// SIMATIC STEP 7 (V5.x) project COB#1&2_GC#2_07_12_2012
// CPU: CPU 315-2 DP
// CPU: CPU 315-2 DP
// station: Hardware
// station: SIMATIC 300 - BEC
// station: P_ADR_BUS
// station: Hardware
// station: SIMATIC 300 - TATA
// station: P_ADR_BUS

SYMBOL_TABLE
"MAIN_POWER_DB"	DB 1	DB 1	// MAIN POWER DATA BLOCK
"HYDRAULIC_FUNCTIONS_DB"	DB 2	DB 2	// HYDRAULIC FUNCTIONS DB
"TRAVEL_DRIVE_DB"	DB 3	DB 3	// TRAVEL DRIVE DATA BLOCK
"AIR_COMPRESSOR_DB"	DB 4	DB 4	// AIR COMPRESSOR DATA BLOCK
"HOOD_SYSTEM_DB"	DB 5	DB 5	// HOOD SYSTEM OPERATIONS DATA BLOCK
"DOOR_EXTRACTOR_DB"	DB 6	DB 6	// DOOR EXTRACTOR MECHANISH DATA BLOCK
"SERVICE_PLATFORM_DB"	DB 7	DB 7	// SERVICE PLATFORM DATA BLOCK
"JAMB_CLEANER_DB"	DB 8	DB 8	// JAMB CLEANER DATA BLOCK
"GUIDE_CAGE_DB"	DB 9	DB 9	// GUIDE CAGE DATA BLOCK
"DOOR_CLEANER_MOTOR_DB"	DB 10	DB 10	// DOOR CLEANER MOTOR DATA BLOCK
"WIN_CC_DB"	DB 11	DB 11	// WIN CC HMI DATA BLOCK
"CMD_FROM_TATA"	DB 12	DB 12	// COMMANDS FROM TATA PLC THROUGH PROFIBUS
"FB_TO_TATA"	DB 13	DB 13	// FEEDBACK TO TATA THROUGH PROFIBUS
"TATA_COMMUNICATION_DB"	DB 14	DB 14	// TATA COMMUNICATION DATA BLOCK
"INPUT_MAPPING"	FC 1	FC 1	// INPUT MAPPING FUNCTION
"OUTPUT_MAPPING"	FC 2	FC 2	// OUTPUT MAPPING FUNCTION
"MAIN_POWER"	FC 3	FC 3	// MAIN POWER CONTROL LOGIC
"HYDRAULIC_SYSTEM"	FC 4	FC 4	// HYDRAULIC SYSTEM OPERATIONS
"TRAVEL_DRIVE"	FC 5	FC 5	// TRAVEL_DRIVE_MECHANISM
"AIR_COMPRESSOR"	FC 6	FC 6	// AIR COMPRESSOR FUNCTION
"HOOD_SYSTEM"	FC 7	FC 7	// HOOD SYSTEM OPERATIONS
"DOOR_EXTRACTOR"	FC 8	FC 8	// DOOR EXTRACTOR MECHANISM
"SERVICE_PLATFORM"	FC 9	FC 9	// SERVICE PLATFORM OPERATIONS
"JAMB_CLEANER"	FC 10	FC 10	// JAMB CLEANER FUNCTIONS
"GUIDE_CAGE"	FC 11	FC 11	// GUIDE CAGE FUNCTION
"DOOR_CLEANER_MOTOR"	FC 12	FC 12	// DOOR CLEANER MOTOR FUNCTIONS
"PROFIBUS_COMMUNICATION"	FC 13	FC 13	// PROFIBUS COMMUNICATION LOGIC
"TATA_COMMUNICATION"	FC 14	FC 14	// TATA COMMUNICATION FUNCATIONS
"SCALE"	FC 105	FC 105	// Scaling Values
"UNSCALE"	FC 106	FC 106	// Unscaling Values
"MAIN_PWR_RDY_FOR_ON"	I 0.0	BOOL	// MAIN POWER READY FOR ON
"MAIN_PWR_ON_FB"	I 0.1	BOOL	// MAIN POWER ON FEED BACK
"CTRL_PWR_ON_FB"	I 0.2	BOOL	// CONTROL POWER ON FEEDBACK
"MAIN_PWR_ON_PB"	I 0.3	BOOL	// MAIN POWER ON PUSH BUTTON
"MAIN_PWR_OFF_PB"	I 0.4	BOOL	// MAIN POWER OFF PUSH BUTTON
"LAMP_TEST_PB"	I 0.5	BOOL	// LAMP TEST PUSH BUTTON
"ALARM_ACK_PB"	I 0.6	BOOL	// ALARM ACKNOWLEDGE PUSH BUTTON
"SERVICE_PF_STP_PB"	I 0.7	BOOL	// SERVICE PLATFORM STOP PUSH BUTTON
"CTRL_SELECTION_CD"	I 1.0	BOOL	// CONTROL SELECTRION CD
"EXT_OVN_DOR_STA_PB"	I 1.1	BOOL	// EXTRACT OVEN DOOR STAT PUSH PUSH BUTTON
"RPL_OVN_DOR_STA_PB"	I 1.2	BOOL	// REPLACE OVEN DOOR STAT PUSH PUSH BUTTON
"EXT_RPL_FUNC_STP_PB"	I 1.3	BOOL	// EXTRACT AND REPLACE FUNCTION STOP PUSH BUTTON
"GC_TRA_AUTO_STA_PB"	I 1.4	BOOL	// GUIDE CAGE TRAVEL AUTO START PUSH BUTTON
"GC_TRA_AUTO_STP_PB"	I 1.5	BOOL	// GUIDE CAGE TRAVEL AUTO STOP PUSH BUTTON
"CLN_OVN_JMB_STA_PB"	I 1.6	BOOL	// CLEAN OVEN JAMB AUTO START PUSH BUTTON
"ALL_OPER_IN_REP_MODE"	I 1.7	BOOL	// ALL OPERATIONS IN REPAIR MODE
"CLN_OVN_JMB_STP_PB"	I 2.0	BOOL	// CLEAN OVEN JAMB AUTO STOP PUSH BUTTON
"ALL_MECH_QUICK_STOP"	I 2.1	BOOL	// ALL MECHANICAL OPERATIONS QUICK STOP
"CLN_OVN_DR_STA_PB"	I 2.2	BOOL	// CLEAN OVEN DOOR START PUSH BUTTON
"CLN_OVN_DR_STP_PB"	I 2.3	BOOL	// CLEAN OVEN DOOR STOP PUSH BUTTON
"CD_EMERGENCY_STOP"	I 2.4	BOOL	// CONTROL DESK EMERGENCY STOP
"SERVICE_PF_STA_PB"	I 2.5	BOOL	// SERVICE PLATFORM START PUSH BUTTON
"REP_MAN_SS"	I 2.6	BOOL	// REPAIR/MANUAL SELECTOR SWITCH
"ALL_OPER_IN_OPER_MODE"	I 2.7	BOOL	// ALL OPERATIONS IN OPERATION MODE
"JC_VC_HM_STA_PB"	I 3.0	BOOL	// JAMB CLEANER HOME START PB
"ID_FAN_READY"	I 3.1	BOOL	// ID FAN DRIVE READY FOR START
"PUMP_1_RUN_FB"	I 3.2	BOOL	// PUMP 1 RUNNING FEEDBACK
"PUMP_1_OVR_LD_TRIP"	I 3.3	BOOL	// PUMP 1 OVER LOAD TRIPPED
"PUMP_2_RDY_FOR_STA"	I 3.4	BOOL	// PUMP 2 READY FOR START
"PUMP_2_RUN_FB"	I 3.5	BOOL	// PUMP 2 RUNNING FEEDBACK
"PUMP_2_OVR_LD_TRIP"	I 3.6	BOOL	// PUMP 2 OVER LOAD TRIPPED
"CIR_PUMP_RDY_FOR_STA"	I 4.0	BOOL	// CIRCULATION PUMP READY FOR START
"CIR_PUMP_RUN_FB"	I 4.1	BOOL	// CIRCULATION PUMP RUNNING FEEDBACK
"CIR_PUMP_OVR_LD_TRIP"	I 4.2	BOOL	// CIRCULATION PUMP OVER LOAD TRIPPED
"COLR_FAN_RDY_FOR_STA"	I 4.3	BOOL	// COOLER FAN READY FOR START
"COLR_FAN_RUN_FB"	I 4.4	BOOL	// COOLER FAN RUNNING FEEDBACK
"COLR_FAN_OVR_LD_TRIP"	I 4.5	BOOL	// COOLER FAN OVER LOAD TRIPPED
"CD_LCS_SS"	I 4.6	BOOL	// CONTROL DESK / LOCAL CONTROL SELECTOR SWITCH
"PUMP_1_2_SS"	I 5.0	BOOL	// PUMP 1 OR 2 SELECTOR SWITCH
"PUMP_1_STA_PB"	I 5.1	BOOL	// PUMP 1 START PUSH BUTTON
"PUMP_1_STP_PB"	I 5.2	BOOL	// PUMP 1 STOP PUSH BUTTON
"PUMP_2_STA_PB"	I 5.3	BOOL	// PUMP 2 START PUSH BUTTON
"PUMP_2_STP_PB"	I 5.4	BOOL	// PUMP 2 STOP PUSH BUTTON
"EMERGENCY_STOP_PB"	I 5.5	BOOL	// EMERGENCY STOP PUSH BUTTON
"LAMP_TEST_PB_LCS_41"	I 5.6	BOOL	// LAMP TEST PUSH BITTON LCS 41
"SP_TRA_FWD_STA_PB"	I 5.7	BOOL	// SERVICE PLATFORM TRAVEL FORWARD PUSH BUTTON
"PUMP_1_2_SS_LCS"	I 6.0	BOOL	// PUMP 1 OR 2 SELECTOR SWITCH LCS
"PUMP_1_STA_PB_LCS"	I 6.1	BOOL	// PUMP 1 START PUSH BUTTON LCS
"PUMP_1_STP_PB_LCS"	I 6.2	BOOL	// PUMP 1 STOP PUSH BUTTON LCS
"PUMP_2_STA_PB_LCS"	I 6.3	BOOL	// PUMP 2 START PUSH BUTTON LCS
"PUMP_2_STP_PB_LCS"	I 6.4	BOOL	// PUMP 2 STOP PUSH BUTTON LCS
"CIR_PUMP_STA_PB_LCS"	I 6.5	BOOL	// CIRCULATION PUMP START PUSH BUTTON LCS
"CIR_PUMP_STP_PB_LCS"	I 6.6	BOOL	// CIRCULATION PUMP STOP PUSH BUTTON LCS
"SP_TRA_REV_STA_PB"	I 6.7	BOOL	// SERVICE PLATFORM TRAVEL REVERSE START PUSH BUTTON
"COLR_FAN_STA_PB_LCS"	I 7.0	BOOL	// COOLER FAN START PUSH BUTTON LCS
"COLR_FAN_STP_PB_LCS"	I 7.1	BOOL	// COOLER FAN STOP PUSH BUTTON LCS
"EMG_ACCM_STA_PB_LCS"	I 7.2	BOOL	// EMERGENCY ACCUMULATOR START PB LCS
"EMG_ACCM_STP_PB_LCS"	I 7.3	BOOL	// EMERGENCY ACCUMULATOR STOP PB LCS
"SHT_OF_VLV_LIN_1_FUL_OPN"	I 7.4	BOOL	// SHUT OFF VALVE IN LINE 1 - FULLY OPEN
"SHT_OF_VLV_LIN_2_FUL_OPN"	I 7.5	BOOL	// SHUT OFF VALVE IN LINE 2 - FULLY OPEN
"LOW_OIL_TEMP"	I 7.6	BOOL	// LOW OIL TEMPERATURE - THERMOSTAT
"SP_STP_PB"	I 7.7	BOOL	// SERVICE PLATFORM STOP PUSH BUTTON
"HIGH_OIL_TEMP"	I 8.0	BOOL	// HIGH OIL TEMPERATURE - THERMOSTAT
"MAX_OIL_TEMP"	I 8.1	BOOL	// MAXIMUM OIL TEMPERATURE - THERMOSTAT
"LOW_OIL_LEVEL"	I 8.2	BOOL	// LOW OIL LEVEL - FLOAT SWITCH
"MIN_OIL_LEVEL"	I 8.3	BOOL	// MINIMUM OIL LEVEL - FLOAT SWITCH
"RET_LIN_FLTR_CKD"	I 8.4	BOOL	// RETURN LINE FILTER CHOKED
"LOW_OIL_PRESS"	I 8.5	BOOL	// LOW OIL PRESSURE - PRESSURE SWITCH
"HIGH_OIL_PRESS"	I 8.6	BOOL	// HIGH OIL PRESSURE - PRESSURE SWITCH
"SP_AUTO_SS"	I 8.7	BOOL	// SERVICE PLATFORM AUTO SELECTOR SWITCH
"TRA_GRP_1_BRK_RDY_FOR_ST"	I 9.0	BOOL	// TRAVEL GROUP 1 BREAK READY FOR START
"TRA_GRP_1_BRK_ON_FB"	I 9.1	BOOL	// TRAVEL GROUP 1 BREAK ON FEEDBACK
"TRA_GRP_2_BRK_RDY_FOR_ST"	I 9.2	BOOL	// TRAVEL GROUP 2 BREAK READY FOR START
"TRA_GRP_2_BRK_ON_FB"	I 9.3	BOOL	// TRAVEL GROUP 2 BREAK ON FEEDBACK
"TRA_JOY_STK_DED_MAN_BTN"	I 9.4	BOOL	// TRAVEL JOY DEAD MAN BUTTON
"TRA_JOY_STK_HME_POS"	I 9.5	BOOL	// TRAVEL JOY STICK HOME POSITION
"TRA_JOY_STK_FWD_POS"	I 9.6	BOOL	// TRAVEL JOY STICK FOWRWARD POSITION
"TRA_JOY_STK_REV_POS"	I 9.7	BOOL	// TRAVEL JOY DEAD REVERSE POSITION
"TRA_MODE_AUTO_MAN_SS"	I 10.0	BOOL	// TRAVEL MODE AUTO/MANUAL BUTTON
"LASER_SPOTTING"	I 10.1	BOOL	// TRAVEL LASER SPOTTING
"AUTO_POS_ACK"	I 10.2	BOOL	// AUTO POSITION ACKNOWLEDGE
"TRA_DRV_1_PROF_HARD_SS"	I 10.3	BOOL	// TRAVEL DRIVE 1 PROFIBUS/HARD WIRE SELECTRO SWITCH
"TRA_DRV_1_ON_FB"	I 10.4	BOOL	// TRAVEL DRIVE 1 ON FEEDBACK
"TRA_DRV_1_RDY_FOR_STA"	I 10.5	BOOL	// TRAVEL DRIVE 1 READY FOR START
"TRA_DRV_1_TRP_FB"	I 10.6	BOOL	// TRAVEL DRIVE 1 TRIP FEEDBACK
"TRA_DRV_2_PROF_HARD_SS"	I 10.7	BOOL	// TRAVEL DRIVE 2 PROFIBUS/HARD WIRE SELECTRO SWITCH
"TRA_DRV_2_ON_FB"	I 11.0	BOOL	// TRAVEL DRIVE 2 ON FEEDBACK
"TRA_DRV_2_RDY_FOR_STA"	I 11.1	BOOL	// TRAVEL DRIVE 2 READY FOR START
"TRA_DRV_2_TRP_FB"	I 11.2	BOOL	// TRAVEL DRIVE 2 TRIP FEEDBACK
"LIMIT_SW_END_FWD_FB"	I 11.3	BOOL	// LIMIT SWITCH END FORWARD FEEDBACK
"LIMIT_SW_END_EMG_FWD_FB"	I 11.4	BOOL	// LIMIT SWITCH END FORWARD EMERGENCY FEEDBACK
"LIMIT_SW_END_REV_FB"	I 11.5	BOOL	// LIMIT SWITCH END REVERSE FEEDBACK
"LIMIT_SW_END_EMG_REV_FB"	I 11.6	BOOL	// LIMIT SWITCH END REVERSE EMERGENCY FEEDBACK
"SP_MAN_SS"	I 11.7	BOOL	// SERVICE PLATFORM MANUAL SELECTOR SWITCH
"SP_TRA_FWD_LS"	I 12.0	BOOL	// SERVICE PLATFORM TRAVEL FORWARD LIMIT SWITCH
"AC_RDY_FOR_STA"	I 12.1	BOOL	// AIR COMPRESSOR READY FOR START
"AC_RUN_FB"	I 12.2	BOOL	// AIR COMPRESSOR RUN FEED BACK
"AC_OLR_TRIP_FB"	I 12.3	BOOL	// AIR COMPRESSOR TRIP FEED BACK
"AC_STA_PB"	I 12.4	BOOL	// AIR COMPRESSOR START PUSH BUTTON
"AC_STP_PB"	I 12.5	BOOL	// AIR COMPRESSOR STOP PUSH BUTTON
"ID_FAN_PROFI_HW_SS"	I 12.6	BOOL	// ID FAN PROFIBUS/HARDWIRE CONNECTION
"SP_TRA_REV_LS"	I 12.7	BOOL	// SERVICE PLATFORM TRAVEL REVERSE LIMIT SWITCH
"ID_FAN_DRV_ON_FB"	I 13.0	BOOL	// ID FAN DRIVE ON FEEDBACK
"ID_FAN_DRV_RDY_FOR_STA"	I 13.1	BOOL	// ID FAN DRIVE READY FOR START
"ID_FAN_DRV_TRIP_FB"	I 13.2	BOOL	// ID FAN DRIVE TRIP FEED BACK
"WTR_PMP_DRV_RDY_FOR_STA"	I 13.3	BOOL	// WATER PUMP DRIVE READY FOR START
"WTR_PMP_DRV_ON_FB"	I 13.4	BOOL	// WATER PUMP DRIVE ON FEEDBACK
"WTR_PMP_DRV_TRIP_FB"	I 13.5	BOOL	// WATER PUMP DRIVE TRIP FEED BACK
"HOOD_STA_PB"	I 13.6	BOOL	// HOOD START PUSH BUTTON
"EMERGENCY_STOP_PB_PANEL"	I 13.7	BOOL	// EMERGENCY STOP PUSH BUTTON IN PLC PANEL
"HOOD_STP_PB"	I 14.0	BOOL	// HOOD STOP PUSH BUTTON
"ID_FAN_LS_HS_SEL"	I 14.1	BOOL	// ID FAN LOW SPEED/HIGH SPEED SELECTION
"WTR_LEV_LOW_LEV_SWH"	I 14.2	BOOL	// WATER LEVEL LOW LEVEL SWITCH
"SLEW_SLOW_FWD_LS"	I 14.3	BOOL	// SLEW SLOW FORWARD LIMIT SWITCH
"SLEW_SLOW_RET_LS"	I 14.4	BOOL	// SLEW SLOW RETRACT LIMIT SWITCH
"SLEW_NOR_FWD_LS"	I 14.5	BOOL	// SLEW NORMAL FORWARD LIMIT SWITCH
"SLEW_NOR_RET_LS"	I 14.6	BOOL	// SLEW NORMAL RETRACT LIMIT SWITCH
"TRA_ILK_BYPASS"	I 14.7	BOOL	// TRAVEL INTERLOCK BYPASS INPUT
"TRA_SLOW_FWD_LS"	I 15.0	BOOL	// TRAVEL SLOW FORWARD LIMIT  SWITCH
"TRA_SLOW_RET_LS"	I 15.1	BOOL	// TRAVEL SLOW RETRACT LIMIT  SWITCH
"TRA_FWD_LS"	I 15.2	BOOL	// TRAVEL FORWARD LIMIT SWIITCH
"TRA_RET_LS"	I 15.3	BOOL	// TRAVEL RETRACT LIMIT SWIITCH
"DOOR_ON_HOOK_LS"	I 15.4	BOOL	// DOOR ON HOOK LIMITSWTCH
"DE_DOOR_LCH_TURN_UP_LS"	I 15.5	BOOL	// DOOR EXTRACTION DOOR LATCH TURNING LOCK LIMIT SWITCH
"DR_LCH_TURN_DN_LS"	I 15.6	BOOL	// DOOR LATCH TURNING DOWN LIMIT SWICH
"LIFT_LDT_TMR_SS"	I 15.7	BOOL	// LIFTING LDT TIMER SELECTOR
"SLEW_FWD_STA_PB"	I 16.0	BOOL	// SLEW FORWARD START PUSH BUTTON
"SLEW_RET_STA_PB"	I 16.1	BOOL	// SLEW RETRACT START
"DOOR_EXT_AUTO_SS"	I 16.2	BOOL	// DOOR EXTRACTOR AUTO SELECTOR SWITCH
"DOOR_EXT_MAN_SS"	I 16.3	BOOL	// DOOR EXTRACTOR MANUAL SELECTOR SWITCH
"DOOR_EXT_STP_PB"	I 16.4	BOOL	// DOOR EXTRACTOR STOP PUSH BUTTON
"VER_COMP_FWD_STA_PB"	I 16.5	BOOL	// VERTICAL COMPENSATION FORWARD START PUSH BUTTON
"VER_COMP_RET_STA_PB"	I 16.6	BOOL	// VERTICAL COMPENSATION RETRACT START PUSH BUTTON
"TRA_FWD_STA_PB"	I 17.0	BOOL	// TRAVEL FORWARD START PUSH BUTTON
"TRA_RET_STA_PB"	I 17.1	BOOL	// TRAVEL RETRACT START PUSH BUTTON
"DR_SPNG_LK_STA_PB"	I 17.2	BOOL	// DOOR SPRING PRESSURE START PUSH BUTTON
"DR_SPNG_UNLK_STA_PB"	I 17.3	BOOL	// DOOR SPRING PRESSURE RELEASE START PUSH BUTTON
"MAIN_STK_UP_STA_PB"	I 17.4	BOOL	// MAIN STROKE UP START PUSH BUTTON
"MAIN_STK_UP_DN_PB"	I 17.5	BOOL	// MAIN STROKE DOWN START PUSH BUTTON
"FIN_STK_UP_STA_PB"	I 17.6	BOOL	// FINAL STROKE UP START PUSH BUTTON
"FIN_STK_DN_PB"	I 18.0	BOOL	// FINAL STROKE DOWN START PUSH BUTTON
"PRE_STK_UP_STA_PB"	I 18.1	BOOL	// PRE STROKE UP START PUSH BUTTON
"PRE_STK_UP_DN_PB"	I 18.2	BOOL	// PRE STROKE DOWN START PUSH BUTTON
"DR_LCH_TURN_UP_PB"	I 18.3	BOOL	// DOOR LATCH TURNING LOCK PUSH BUTTON
"DR_LCH_TURN_DN_PB"	I 18.4	BOOL	// DOOR LATCH TURNING UNLOCK PUSH BUTTON
"AIR_COMMP_PS"	I 18.5	BOOL	// AIR COMMPRESSOR PRESSURE SWITCH
"SERV_PF_FWD_RUN_FB"	I 19.3	BOOL	// SERVICE PLATFORM FORWARD RUN FEED BACK
"SERV_PF_REV_RUN_FB"	I 19.4	BOOL	// SERVICE PLATFORM REVERSE RUN FEED BACK
"SERV_PF_OLR_TRIP_FB"	I 19.5	BOOL	// SERVICE PLATFORM OVERLOAD TRIP FEED BACK
"JC_CAR_TRA_FWD_LS"	I 20.4	BOOL	// JAMB CLEANER CARRIAGE TRAVEL FORWARD LIMIT SWITCH
"JC_CAR_TRA_RET_LS"	I 20.5	BOOL	// JAMB CLEANER CARRIAGE TRAVEL RETRACT LIMIT SWITCH
"JC_VER_CLNR_UP_LS"	I 20.6	BOOL	// JAMB CLEANER VERTICAL CLEANER UP LIMIT SWITCH
"JC_VER_CLNR_DN_LS"	I 21.0	BOOL	// JAMB CLEANER VERTICAL CLEANER DOWN LIMIT SWITCH
"JC_VER_CLNR_HME_LS"	I 21.1	BOOL	// JAMB CLEANER VERTICAL CLEANER HOME LIMIT SWITCH
"JC_CRA_TRA_FWD_STA_PB"	I 21.2	BOOL	// JAMB CLEANER CARRIAGE TRAVEL FORWARD PUSH BUTTON
"JC_CRA_TRA_RET_STA_PB"	I 21.3	BOOL	// JAMB CLEANER CARRIAGE TRAVEL RETRACT PUSH BUTTON
"JC_VER_CLNR_UP_STA_PB"	I 21.4	BOOL	// JAMB CLEANER VERTICAL CLEANER UP START PUSH BUTTON
"JC_VER_CLNR_DN_STA_PB"	I 21.5	BOOL	// JAMB CLEANER VERTICAL CLEANER DOWN START PUSH BUTTON
"JC_STP_PB"	I 21.6	BOOL	// JAMB CLEANER OPERATIONS STOP PUSH BUTTON
"JC_AUTO_MAN_SS"	I 22.0	BOOL	// JAMB CLEANER AUTO MANUAL SELECTOR SWITCH
"GC_TRA_FWD_LS"	I 22.1	BOOL	// GUIDE CAGE TRAVEL FORWARD LIMIT SWITCH
"GC_TRA_RET_LS"	I 22.2	BOOL	// GUIDE CAGE TRAVEL RETRACT LIMIT SWITCH
"GC_AUTO_SS"	I 22.3	BOOL	// GUIDE CAGE AUTO SELECTOR SWITCH
"GC_MAN_SS"	I 22.4	BOOL	// GUIDE CAGE MANUAL SELECTOR SWITCH
"GC_TRA_FWD_STA_PB"	I 22.5	BOOL	// GUIDE CAGE TRAVEL FORWARD START PUSH BUTTON
"GC_TRA_RET_STA_PB"	I 22.6	BOOL	// GUIDE CAGE TRAVEL RETRACT START PUSH BUTTON
"GC_STP_PB"	I 23.0	BOOL	// GUIDE CAGE AUTO STOP PUSH BUTTON
"DC_RDY_FOR_STA"	I 23.1	BOOL	// DOOR CLEANER READY FOR START
"DC_UP_RUN_FB"	I 23.2	BOOL	// DOOR CLEANER UP RUNNING FEED BACK
"DC_OLR_TRIP"	I 23.3	BOOL	// DOOR CLEANER OVER LOAD TRIP
"DC_DN_RUN_FB"	I 23.4	BOOL	// DOOR CLEANER DOWN RUNNING FEED BACK
"DC_AUTO_SS"	I 23.5	BOOL	// DOOR CLEANER AUTO SELECTOR SWITCH
"DC_MAN_SS"	I 23.6	BOOL	// DOOR CLEANER MANUAL SELECTOR SWITCH
"DC_UP_STA_PB"	I 24.0	BOOL	// DOOR CLEANER UP START PUSH BUTTON
"DC_DN_STA_PB"	I 24.1	BOOL	// DOOR CLEANER DOWN START PUSH BUTTON
"DC_STP_PB"	I 24.2	BOOL	// DOOR CLEANER STOP PUSH BUTTON
"DC_HME_PB"	I 24.3	BOOL	// DOOR CLEANER HOME PUSH BUTTON
"DC_UP_LS"	I 24.4	BOOL	// DOOR CLEANER UP LIMIT SWITCH
"DC_DN_LS"	I 24.5	BOOL	// DOOR CLEANER DOWN LIMIT SWITCH
"DC_HME_LS"	I 24.6	BOOL	// DOOR CLEANER HOME LIMIT SWITCH
"ALWAYS_OFF"	M 0.0	BOOL	// BIT WILL BE ALWAYS OFF
"ALWAYS_ON"	M 0.1	BOOL	// THIS BIT WILL BE ALWAYS ON
"HALF_SECOND_PULSE_TRAIN"	M 0.2	BOOL	// THIS BIT WILL BE ON FOR 500MS AND OFF FOR 500MS
"ONE_SECOND_PULSE"	M 0.3	BOOL	// THIS BIT WILL BE HIGH ON THE RAISING EDGE OF M0.2
"EMERGENCY"	M 0.4	BOOL	// EMERGENCY PRESSED
"PULSE_GENERATION_BIT"	M 0.5	BOOL	// THIS BIT IS USED TO GENERATE RAISING EDGE PULSE
"MAIN_PROGRAM"	OB 1	OB 1	// MAIN CYCLIC PROGRAM
"I/O_FLT1"	OB 82	OB 82	// I/O Point Fault 1
"RACK_FLT"	OB 86	OB 86	// Loss of Rack Fault
"PROG_ERR"	OB 121	OB 121	// Programming Error
"MOD_ERR"	OB 122	OB 122	// Module Access Error
"TRA_SPD_REF_VAL_FRM_JS"	PIW 254	INT	// TRAVEL SPEED REFERENCE VALUE FROM JOY STICK
"MAIN_PWR_ON_CMD"	Q 0.0	BOOL	// MAIN POWER ON COMMAND
"MAIN_PWR_ON_IND"	Q 0.1	BOOL	// MAIN POWER ON INDICATOR
"CTRL_PWR_ON_IND"	Q 0.2	BOOL	// CONTROL POWER ON INDICATOR
"SERVICE_PF_IND"	Q 0.3	BOOL	// SERVICE PLATFORM INDICATOR
"FIN_OVN_DOR_IND"	Q 0.4	BOOL	// FINISH OVEN DOOR INDICATOR
"EXT_OVN_DOR_IND"	Q 0.5	BOOL	// EXTRACT OVEN DOOR INDICATOR
"RPL_OVN_DOR_IND"	Q 0.6	BOOL	// REPLACE OVEN DOOR INDICATOR
"LT_SIREN"	Q 0.7	BOOL	// LONG TRAVEL SIREN
"GC_TRA_AUTO_IND"	Q 1.0	BOOL	// GUIDE CAGE AUTO OPERATION INDICATOR
"CLN_OVN_JMB_IND"	Q 1.1	BOOL	// CLEAN OVEN JAMB AUTO INDICATOR
"CLN_OVN_DR_AUTO_IND"	Q 1.2	BOOL	// CLEAN OVEN DOOR AUTO INDICATOR
"PUMP_1_ON_CMD"	Q 1.3	BOOL	// PUMP 1 ON COMMAND
"PUMP_2_ON_CMD"	Q 1.4	BOOL	// PUMP 2 ON COMMAND
"CIR_PUMP_ON_CMD"	Q 1.5	BOOL	// CIRCULATION PUMP ON COMMAND
"CLR_FAN_ON_CMD"	Q 1.6	BOOL	// COOLER FAN ON COMMAND
"GC_PERM"	Q 1.7	BOOL	// GUIDE CAGE PERMISSION
"SYSTEM_RDY_IND"	Q 2.0	BOOL	// SYSTEM READY INDICATOR
"PUMP_1_ON_IND"	Q 2.1	BOOL	// PUMP 1 ON INDICATOR
"PUMP_2_ON_IND"	Q 2.2	BOOL	// PUMP 2 ON INDICATOR
"LOCAL_ON_IND_LCS_41"	Q 2.3	BOOL	// LCS - 41 LOCAL ON INDICATOR
"HIGH_OIL_TEMP_IND_LCS"	Q 2.4	BOOL	// HIGH OIL TEMPERATURE INDICATOR LCS
"LOW_OIL_LEVEL_IND_LCS"	Q 2.5	BOOL	// LOW OIL LEVEL INDICATOR LCS
"LOW_OIL_TEMP_IND_LCS"	Q 2.6	BOOL	// LOW OIL TEMPERATURE INDICATOR LCS
"FLTR_CHK_IND_LCS"	Q 3.0	BOOL	// FILTER CHOKE INDICATOR LCS
"PUMP_1_ON_IND_LCS"	Q 3.1	BOOL	// PUMP 1 ON INDICATOR LCS
"PUMP_2_ON_IND_LCS"	Q 3.2	BOOL	// PUMP 2 ON INDICATOR LCS
"CIR_PUMP_ON_IND_LCS"	Q 3.3	BOOL	// CIRCULATION PUMP ON INDICATOR LCS
"CLR_FAN_ON_IND_LCS"	Q 3.4	BOOL	// COOLER FAN ON INDICATOR LCS
"ACCM_IN_OPER_IND_LCS"	Q 3.5	BOOL	// ACCUMULATOR IN OPERATION INDICATOR
"PRESS_REL_VLV_1_ON_CMD"	Q 4.0	BOOL	// PRESSURE RELIEF VALVE 1 ON COMMAND
"PRESS_REL_VLV_2_ON_CMD"	Q 4.1	BOOL	// PRESSURE RELIEF VALVE 2 ON COMMAND
"EMG_ACCM_ON_CMD"	Q 4.2	BOOL	// EMERGENCY ACCUMULLATOR ON COMMAND
"TRA_BRK_1_ON_CMD"	Q 4.3	BOOL	// TRAVEL GROUP 1 BRAKE ON COMMAND
"TRA_BRK_2_ON_CMD"	Q 4.4	BOOL	// TRAVEL GROUP 2 BRAKE ON COMMAND
"TRA_PER_IND"	Q 4.5	BOOL	// TRAVEL PERMISSION INDICATOR
"AUTO_POS_ON"	Q 4.6	BOOL	// AUTO POSITION ON
"TRA_DRV_1_ON_CMD"	Q 4.7	BOOL	// TRAVEL DRIVE 1 ON COMMAND
"TRA_DRV_1_FWD_CMD"	Q 5.0	BOOL	// TRAVEL DRIVE 1 FORWARD COMMAND
"TRA_DRV_1_REV_CMD"	Q 5.1	BOOL	// TRAVEL DRIVE 1 REVERSE COMMAND
"TRA_DRV_2_ON_CMD"	Q 5.2	BOOL	// TRAVEL DRIVE 2 ON COMMAND
"TRA_DRV_2_FWD_CMD"	Q 5.3	BOOL	// TRAVEL DRIVE 2 FORWARD COMMAND
"TRA_DRV_2_REV_CMD"	Q 5.4	BOOL	// TRAVEL DRIVE 2 REVERSE COMMAND
"AC_ON_CMD"	Q 5.6	BOOL	// AIR COMPRESSOR ON COMMAND
"AC_ON_IND"	Q 6.0	BOOL	// AIR COMPRESSOR ON INDICATOR
"ID_FAN_HIGH_SPD_CMD"	Q 6.1	BOOL	// ID FAN HIGH SPEED COMMAND
"ID_FAN_LOW_SPD_CMD"	Q 6.2	BOOL	// ID FAN LOW SPEED COMMAND
"ID_FAN_REV_ON_CMD"	Q 6.3	BOOL	// ID FAN REVERSE ON COMMADN COMMAND
"WTR_PMP_ON_CMD"	Q 6.4	BOOL	// WATER PUMP ON COMMAND
"HOOD_ON_IND"	Q 6.5	BOOL	// HOOD ON INDICATOR
"SLEW_SLOW_RET_CMD"	Q 6.6	BOOL	// SLEW SLOW RETRACT COMMAND
"SLEW_NOR_FWD_COMMAND"	Q 7.0	BOOL	// SLEW NORMAL FORWARD COMMAND
"SLEW_NOR_RET_COMMAND"	Q 7.1	BOOL	// SLEW NORMAL RETRACT COMMAND
"VER_COMP_FWD_CMD"	Q 7.2	BOOL	// VERTICAL COMPENSATION FORWARD COMMAND
"VER_COMP_RET_CMD"	Q 7.3	BOOL	// VERTICAL COMPENSATION RETRACT COMMAND
"VER_COMP_RELIVE_CMD"	Q 7.4	BOOL	// VERTICAL COMPENSTAION RELIVE  COOMMAND
"TRA_SLOW_FWD_CMD"	Q 7.5	BOOL	// TRAVEL SLOW FORWARD COMMAND
"TRA_SLOW_RET_CMD"	Q 7.6	BOOL	// TRAVEL SLOW RETRACT COMMAND
"TRA_NOR_FWD_CMD"	Q 8.0	BOOL	// TRAVEL NORMAL FORWARD COMMAND
"TRA_NOR_RET_CMD"	Q 8.1	BOOL	// TRAVEL NORMAL RETRACT COMMAND
"TRA_RELIVE_CMD"	Q 8.2	BOOL	// TRAVEL RELIVE COOMMAND
"DR_SPNG_LK_CMD"	Q 8.3	BOOL	// DOOR SPRING PRESS LOCK COMMAND
"DR_SPNG_UNLK_CMD"	Q 8.4	BOOL	// DOOR SPRING PRESS UNLOCK COMMAND
"MAIN_STK_UP_CMD"	Q 8.5	BOOL	// MAIN STROKE UP COMMAND
"MAIN_STK_DN_CMD"	Q 8.6	BOOL	// MAIN STROKE DN COMMAND
"PRE_STK_UP_CMD"	Q 9.0	BOOL	// PRE STROKE UP COMMAND
"PRE_STK_DN_CMD"	Q 9.1	BOOL	// PRE STROKE DN COMMAND
"DR_LCH_TURN_UP_CMD"	Q 9.2	BOOL	// DOOR LATCH TURNING UP COMMAND
"DR_LCH_TURN_DN_CMD"	Q 9.3	BOOL	// DOOR LATCH TURNING DOWN COMMADN
"SLEW_SLOW_FWD_CMD"	Q 9.4	BOOL	// SLEW SLOW FORWARD COMMAND
"DE_DR_LCH_TURN_UP_IND"	Q 9.5	BOOL	// DOOR EXTRACTION DOOR LATCH TURNING LOCK INDICATOR
"DR_LCH_TURN_DN_IND"	Q 9.6	BOOL	// DOOR EXTRACTION DOOR LATCH UNLOCK INDICATOR
"SLEW_SLOW_FWD_IND"	Q 10.0	BOOL	// SLEW SLOW FORWARD INDICATOR
"SLEW_SLOW_RET_IND"	Q 10.1	BOOL	// SLEW SLOW RETRACT INDICATOR
"VER_COMP_FWD_IND"	Q 10.2	BOOL	// VERTICAL COMPENSATION FORWARD INDICATOR
"VER_COMP_RET_IND"	Q 10.3	BOOL	// VERTICAL COMPENSATION RETRACT INDICATOR
"TRA_FWD_IND"	Q 10.4	BOOL	// TRAVEL FORWARD INDICATOR
"TRA_RET_IND"	Q 10.5	BOOL	// TRAVEL BACK INDICATOR
"MAIN_STK_UP_IND"	Q 10.6	BOOL	// MAIN STROKE  UP INDICATION
"MAIN_STK_DN_IND"	Q 11.0	BOOL	// MAIN STROKE  DOWN  INDICATOR
"FIN_STK_UP_IND"	Q 11.1	BOOL	// FINAL STROKE  UP INDICATOR
"FIN_STK_DN_IND"	Q 11.2	BOOL	// FINAL STROKE  DOWN INDICATOR
"PRE_STK_UP_IND"	Q 11.3	BOOL	// PRE STROKE  UP INDICATION
"PRE_STK_DN_IND"	Q 11.4	BOOL	// PRE STROKE  DOWN INDICATOR
"DR_SPNG_LK_IND"	Q 11.5	BOOL	// DOOR SPRING PRESS LOCK INDICATOR
"DR_SPNG_UNLK_IND"	Q 11.6	BOOL	// DOOR SPRING PRESS UNLOCK INDICATOR
"SP_TRA_FWD_CMD"	Q 12.0	BOOL	// SERVICE PLATFORM TRAVEL FORWARD START COMMAND
"SP_TRA_REV_CMD"	Q 12.1	BOOL	// SERVICE PLATFORM RETRACT START COMMAND
"LT_ALARM"	Q 12.2	BOOL	// LONG TRAVEL ALARM
"SP_TRA_FWD_IND"	Q 12.4	BOOL	// SERVICE PLATFORM FORWARD INDICATOR
"SP_TRA_RET_IND"	Q 12.5	BOOL	// SERVICE PLATFORM RETRACT INDICATOR
"JC_CAR_TRA_FWD_CMD"	Q 13.1	BOOL	// JAMB CLEANER CARRIAGE TRAVEL FORWARD COMMAND
"JC_CAR_TRA_RET_CMD"	Q 13.2	BOOL	// JAMB CLEANER CARRIAGE TRAVEL RETRACT COMMAND
"JC_VER_CLNR_UP_CMD"	Q 13.3	BOOL	// JAMB CLEANER VERTICAL CLEANER UP COMMAND
"JC_VER_CLNR_DN_CMD"	Q 13.4	BOOL	// JAMB CLEANER VERTICAL CLEANER DOWN COMMAND
"JC_CAR_TRA_FWD_IND"	Q 13.5	BOOL	// JAMB CLEANER CARRIAGE TRAVEL FORWARD INDICATOR
"JC_CAR_TRA_RET_IND"	Q 13.6	BOOL	// JAMB CLEANER CARRIAGE TRAVEL RETRACT INDICATOR
"JC_VER_CLNR_UP_IND"	Q 14.0	BOOL	// JAMB CLEANER VERTICAL CLEANER UP INDICATOR
"JC_VER_CLNR_DN_IND"	Q 14.1	BOOL	// JAMB CLEANER VERTICAL CLEANER DOWN INDICATOR
"JC_VER_CLNR_HME_IND"	Q 14.2	BOOL	// JAMB CLEANER VERTICAL CLEANER HOME INDIATOR
"GC_TRA_FWD_CMD"	Q 14.3	BOOL	// GUIDE CAGE TRAVEL FORWARD COMMAND
"GC_TRA_RET_CMD"	Q 14.4	BOOL	// GUIDE CAGE TRAVEL RETRACT COMMAND
"GC_TRA_FWD_IND"	Q 14.5	BOOL	// GUIDE CAGE TRAVEL FORWARD INDICATOR
"GC_TRA_RET_IND"	Q 14.6	BOOL	// GUIDE CAGE TRAVEL RETRACT INDICATOR
"DC_UP_ON_CMD"	Q 15.0	BOOL	// DOOR CLEANER UP ON COMMAND
"DC_DN_ON_CMD"	Q 15.1	BOOL	// DOOR CLEANER DOWN ON COMMADN
"DC_UP_IND"	Q 15.2	BOOL	// DOOR CLEANER UP INDICATOR
"DC_DN_IND"	Q 15.3	BOOL	// DOOR CLEANER DOWN INDICATOR
"DC_HME_IND"	Q 15.4	BOOL	// DOOR CLEANER HOME INDICATOR
"DPRD_DAT"	SFC 14	SFC 14	// Read Consistent Data of a Standard DP Slave
"DPWR_DAT"	SFC 15	SFC 15	// Write Consistent Data to a Standard DP Slave
"MAIN_STK_UP_CMD_TIM_BAS"	T 20	TIMER	// MAIN STROKE UP COMMAND CUT TIMER BASED
"MAIN_STK_DN_CMD_TIM_BAS"	T 21	TIMER	// MAIN STROKE DOWN COMMAND CUT TIMER BASED
"FIN_STK_DN_CMD_TIM_BAS"	T 22	TIMER	// FINAL STROKE DOWN COMMAND CUT TIMER BASED
"FIN_STK_UP_CMD_TIM_BAS"	T 23	TIMER	// FINAL STROKE UP COMMAND CUT TIMER BASED
"PRE_STK_UP_CMD_TIM_BAS"	T 24	TIMER	// PRE STROKE UP COMMAND CUT TIMER BASED
"PRE_STK_DN_CMD_TIM_BAS"	T 25	TIMER	// PRE STROKE DOWN COMMAND CUT TIMER BASED
"VER_COMP_FWD_LDT_TMR"	T 50	TIMER	// VERTICAL COMPENSATION FORWARD LDT TIMER
"VER_COMP_RET_LDT_TMR"	T 51	TIMER	// VERTICAL COMPENSATION RETRACT LDT TIMER
"VAT_PIW_LDT"	VAT 1	
"VAT_2"	VAT 2	
END_SYMBOL_TABLE

FUNCTION "INPUT_MAPPING" : VOID	// FC 1
AUTHOR : Kamillas
VERSION : 0.1
BEGIN
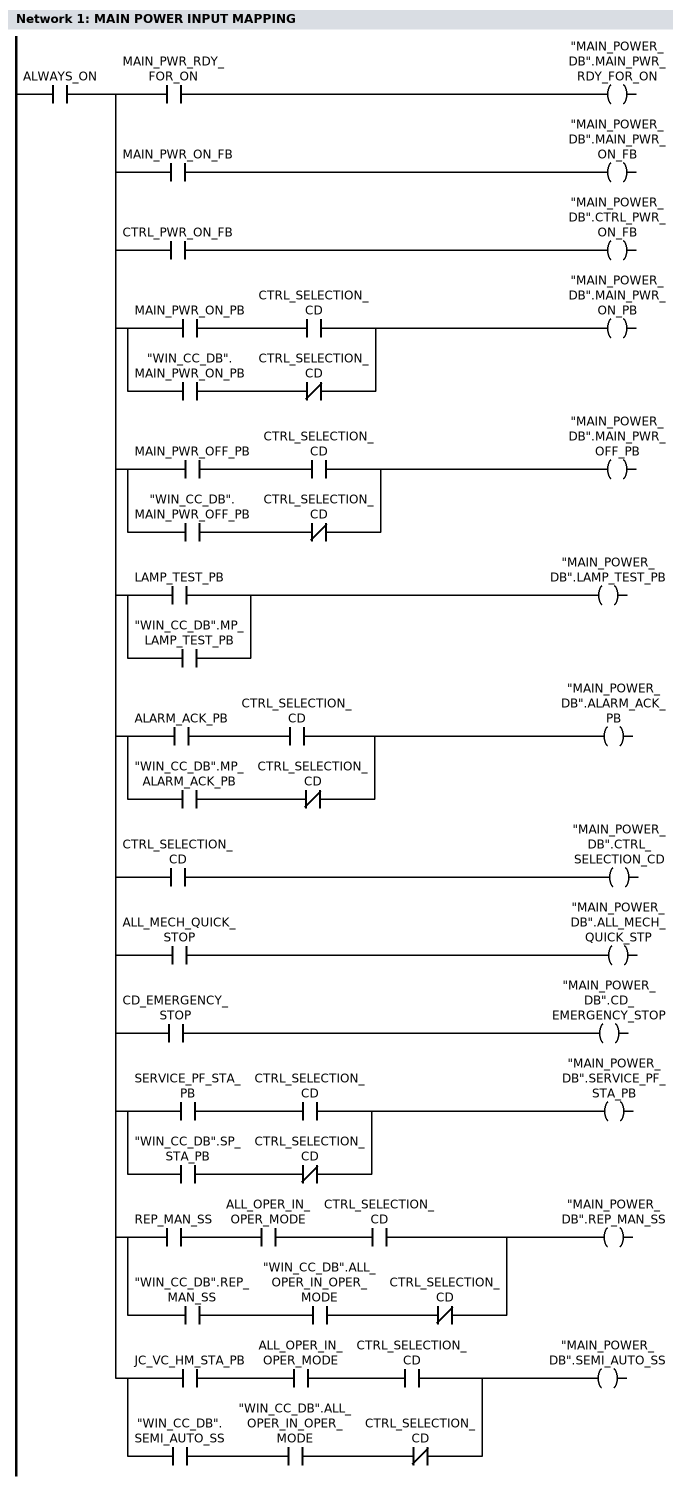
NETWORK
TITLE = MAIN POWER INPUT MAPPING
      A     "ALWAYS_ON";
      =     L 0.0;
      A     L 0.0;
      A     "MAIN_PWR_RDY_FOR_ON";
      =     "MAIN_POWER_DB".MAIN_PWR_RDY_FOR_ON;
      A     L 0.0;
      A     "MAIN_PWR_ON_FB";
      =     "MAIN_POWER_DB".MAIN_PWR_ON_FB;
      A     L 0.0;
      A     "CTRL_PWR_ON_FB";
      =     "MAIN_POWER_DB".CTRL_PWR_ON_FB;
      A     L 0.0;
      A(;
      A     "MAIN_PWR_ON_PB";
      A     "CTRL_SELECTION_CD";
      O;
      A     "WIN_CC_DB".MAIN_PWR_ON_PB;
      AN    "CTRL_SELECTION_CD";
      );
      =     "MAIN_POWER_DB".MAIN_PWR_ON_PB;
      A     L 0.0;
      A(;
      A     "MAIN_PWR_OFF_PB";
      A     "CTRL_SELECTION_CD";
      O;
      A     "WIN_CC_DB".MAIN_PWR_OFF_PB;
      AN    "CTRL_SELECTION_CD";
      );
      =     "MAIN_POWER_DB".MAIN_PWR_OFF_PB;
      A     L 0.0;
      A(;
      O     "LAMP_TEST_PB";
      O     "WIN_CC_DB".MP_LAMP_TEST_PB;
      );
      =     "MAIN_POWER_DB".LAMP_TEST_PB;
      A     L 0.0;
      A(;
      A     "ALARM_ACK_PB";
      A     "CTRL_SELECTION_CD";
      O;
      A     "WIN_CC_DB".MP_ALARM_ACK_PB;
      AN    "CTRL_SELECTION_CD";
      );
      =     "MAIN_POWER_DB".ALARM_ACK_PB;
      A     L 0.0;
      A     "CTRL_SELECTION_CD";
      =     "MAIN_POWER_DB".CTRL_SELECTION_CD;
      A     L 0.0;
      A     "ALL_MECH_QUICK_STOP";
      =     "MAIN_POWER_DB".ALL_MECH_QUICK_STP;
      A     L 0.0;
      A     "CD_EMERGENCY_STOP";
      =     "MAIN_POWER_DB".CD_EMERGENCY_STOP;
      A     L 0.0;
      A(;
      A     "SERVICE_PF_STA_PB";
      A     "CTRL_SELECTION_CD";
      O;
      A     "WIN_CC_DB".SP_STA_PB;
      AN    "CTRL_SELECTION_CD";
      );
      =     "MAIN_POWER_DB".SERVICE_PF_STA_PB;
      A     L 0.0;
      A(;
      A     "REP_MAN_SS";
      A     "ALL_OPER_IN_OPER_MODE";
      A     "CTRL_SELECTION_CD";
      O;
      A     "WIN_CC_DB".REP_MAN_SS;
      A     "WIN_CC_DB".ALL_OPER_IN_OPER_MODE;
      AN    "CTRL_SELECTION_CD";
      );
      =     "MAIN_POWER_DB".REP_MAN_SS;
      A     L 0.0;
      A(;
      A     "JC_VC_HM_STA_PB";
      A     "ALL_OPER_IN_OPER_MODE";
      A     "CTRL_SELECTION_CD";
      O;
      A     "WIN_CC_DB".SEMI_AUTO_SS;
      A     "WIN_CC_DB".ALL_OPER_IN_OPER_MODE;
      AN    "CTRL_SELECTION_CD";
      );
      =     "MAIN_POWER_DB".SEMI_AUTO_SS;
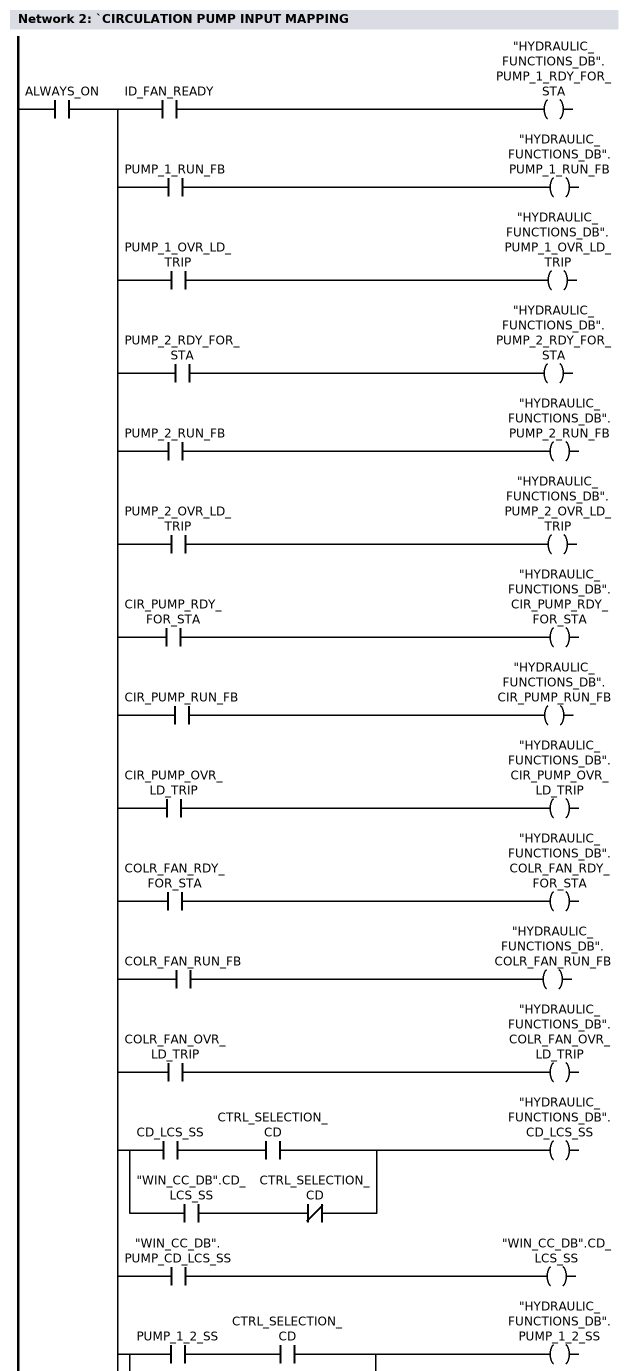
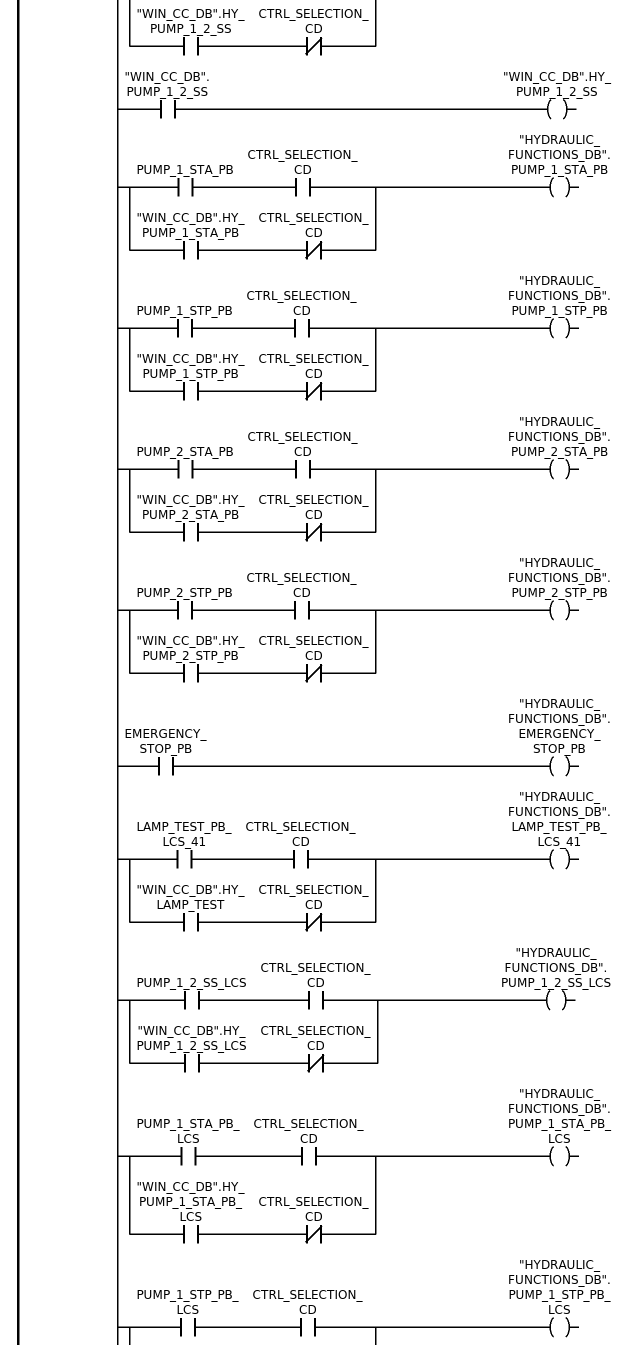
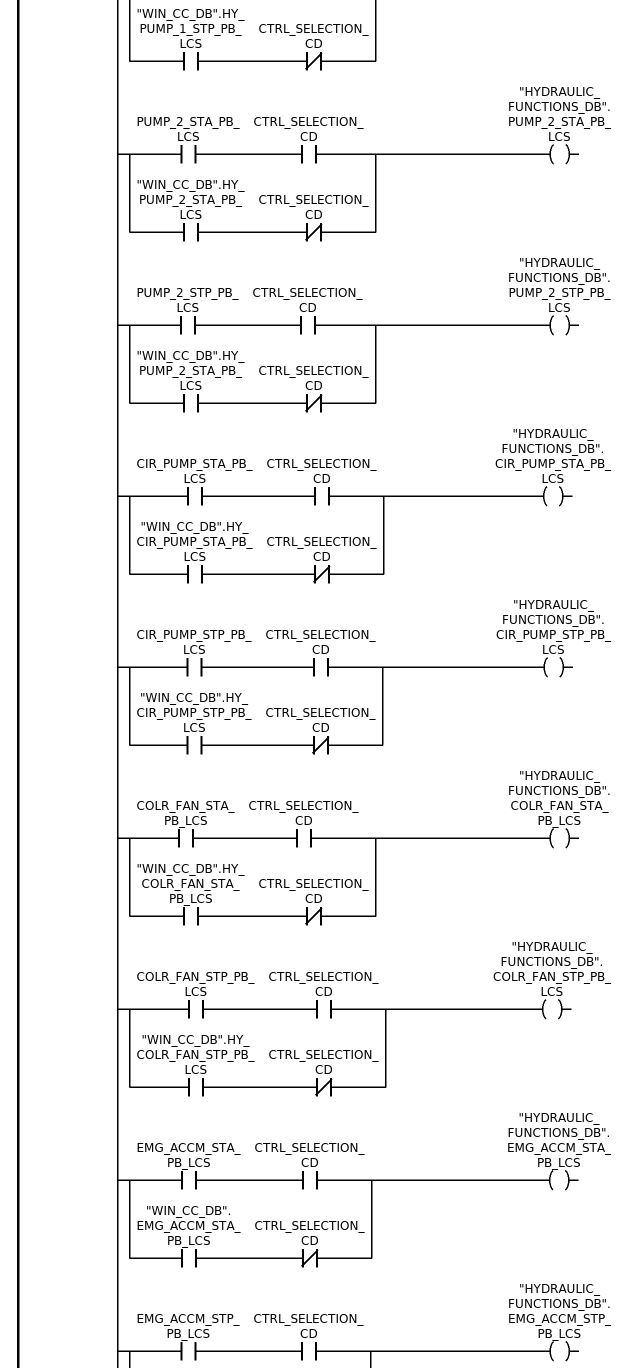
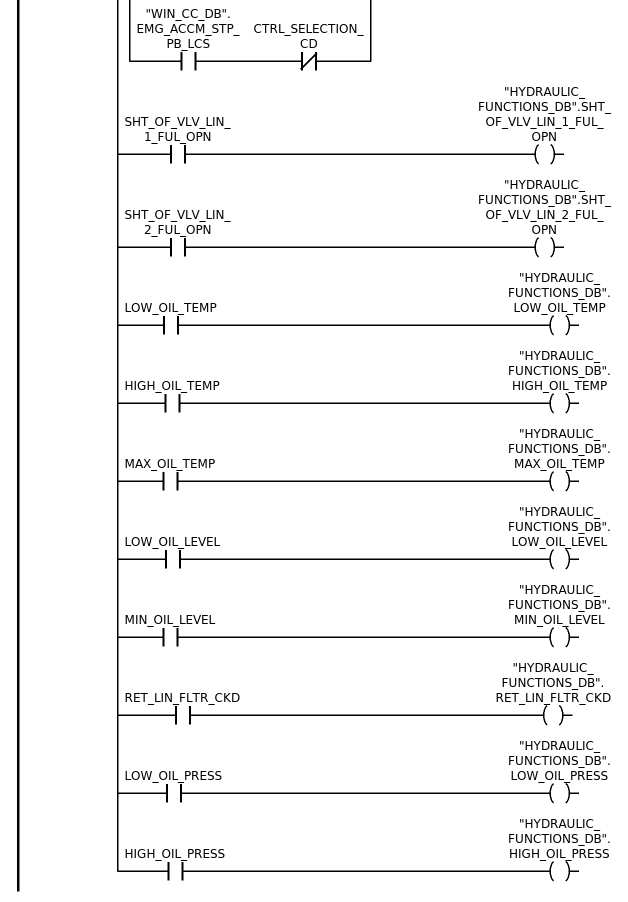
NETWORK
TITLE = `CIRCULATION PUMP INPUT MAPPING
      A     "ALWAYS_ON";
      =     L 0.0;
      A     L 0.0;
      A     "ID_FAN_READY";
      =     "HYDRAULIC_FUNCTIONS_DB".PUMP_1_RDY_FOR_STA;
      A     L 0.0;
      A     "PUMP_1_RUN_FB";
      =     "HYDRAULIC_FUNCTIONS_DB".PUMP_1_RUN_FB;
      A     L 0.0;
      A     "PUMP_1_OVR_LD_TRIP";
      =     "HYDRAULIC_FUNCTIONS_DB".PUMP_1_OVR_LD_TRIP;
      A     L 0.0;
      A     "PUMP_2_RDY_FOR_STA";
      =     "HYDRAULIC_FUNCTIONS_DB".PUMP_2_RDY_FOR_STA;
      A     L 0.0;
      A     "PUMP_2_RUN_FB";
      =     "HYDRAULIC_FUNCTIONS_DB".PUMP_2_RUN_FB;
      A     L 0.0;
      A     "PUMP_2_OVR_LD_TRIP";
      =     "HYDRAULIC_FUNCTIONS_DB".PUMP_2_OVR_LD_TRIP;
      A     L 0.0;
      A     "CIR_PUMP_RDY_FOR_STA";
      =     "HYDRAULIC_FUNCTIONS_DB".CIR_PUMP_RDY_FOR_STA;
      A     L 0.0;
      A     "CIR_PUMP_RUN_FB";
      =     "HYDRAULIC_FUNCTIONS_DB".CIR_PUMP_RUN_FB;
      A     L 0.0;
      A     "CIR_PUMP_OVR_LD_TRIP";
      =     "HYDRAULIC_FUNCTIONS_DB".CIR_PUMP_OVR_LD_TRIP;
      A     L 0.0;
      A     "COLR_FAN_RDY_FOR_STA";
      =     "HYDRAULIC_FUNCTIONS_DB".COLR_FAN_RDY_FOR_STA;
      A     L 0.0;
      A     "COLR_FAN_RUN_FB";
      =     "HYDRAULIC_FUNCTIONS_DB".COLR_FAN_RUN_FB;
      A     L 0.0;
      A     "COLR_FAN_OVR_LD_TRIP";
      =     "HYDRAULIC_FUNCTIONS_DB".COLR_FAN_OVR_LD_TRIP;
      A     L 0.0;
      A(;
      A     "CD_LCS_SS";
      A     "CTRL_SELECTION_CD";
      O;
      A     "WIN_CC_DB".CD_LCS_SS;
      AN    "CTRL_SELECTION_CD";
      );
      =     "HYDRAULIC_FUNCTIONS_DB".CD_LCS_SS;
      A     L 0.0;
      A     "WIN_CC_DB".PUMP_CD_LCS_SS;
      =     "WIN_CC_DB".CD_LCS_SS;
      A     L 0.0;
      A(;
      A     "PUMP_1_2_SS";
      A     "CTRL_SELECTION_CD";
      O;
      A     "WIN_CC_DB".HY_PUMP_1_2_SS;
      AN    "CTRL_SELECTION_CD";
      );
      =     "HYDRAULIC_FUNCTIONS_DB".PUMP_1_2_SS;
      A     L 0.0;
      A     "WIN_CC_DB".PUMP_1_2_SS;
      =     "WIN_CC_DB".HY_PUMP_1_2_SS;
      A     L 0.0;
      A(;
      A     "PUMP_1_STA_PB";
      A     "CTRL_SELECTION_CD";
      O;
      A     "WIN_CC_DB".HY_PUMP_1_STA_PB;
      AN    "CTRL_SELECTION_CD";
      );
      =     "HYDRAULIC_FUNCTIONS_DB".PUMP_1_STA_PB;
      A     L 0.0;
      A(;
      A     "PUMP_1_STP_PB";
      A     "CTRL_SELECTION_CD";
      O;
      A     "WIN_CC_DB".HY_PUMP_1_STP_PB;
      AN    "CTRL_SELECTION_CD";
      );
      =     "HYDRAULIC_FUNCTIONS_DB".PUMP_1_STP_PB;
      A     L 0.0;
      A(;
      A     "PUMP_2_STA_PB";
      A     "CTRL_SELECTION_CD";
      O;
      A     "WIN_CC_DB".HY_PUMP_2_STA_PB;
      AN    "CTRL_SELECTION_CD";
      );
      =     "HYDRAULIC_FUNCTIONS_DB".PUMP_2_STA_PB;
      A     L 0.0;
      A(;
      A     "PUMP_2_STP_PB";
      A     "CTRL_SELECTION_CD";
      O;
      A     "WIN_CC_DB".HY_PUMP_2_STP_PB;
      AN    "CTRL_SELECTION_CD";
      );
      =     "HYDRAULIC_FUNCTIONS_DB".PUMP_2_STP_PB;
      A     L 0.0;
      A     "EMERGENCY_STOP_PB";
      =     "HYDRAULIC_FUNCTIONS_DB".EMERGENCY_STOP_PB;
      A     L 0.0;
      A(;
      A     "LAMP_TEST_PB_LCS_41";
      A     "CTRL_SELECTION_CD";
      O;
      A     "WIN_CC_DB".HY_LAMP_TEST;
      AN    "CTRL_SELECTION_CD";
      );
      =     "HYDRAULIC_FUNCTIONS_DB".LAMP_TEST_PB_LCS_41;
      A     L 0.0;
      A(;
      A     "PUMP_1_2_SS_LCS";
      A     "CTRL_SELECTION_CD";
      O;
      A     "WIN_CC_DB".HY_PUMP_1_2_SS_LCS;
      AN    "CTRL_SELECTION_CD";
      );
      =     "HYDRAULIC_FUNCTIONS_DB".PUMP_1_2_SS_LCS;
      A     L 0.0;
      A(;
      A     "PUMP_1_STA_PB_LCS";
      A     "CTRL_SELECTION_CD";
      O;
      A     "WIN_CC_DB".HY_PUMP_1_STA_PB_LCS;
      AN    "CTRL_SELECTION_CD";
      );
      =     "HYDRAULIC_FUNCTIONS_DB".PUMP_1_STA_PB_LCS;
      A     L 0.0;
      A(;
      A     "PUMP_1_STP_PB_LCS";
      A     "CTRL_SELECTION_CD";
      O;
      A     "WIN_CC_DB".HY_PUMP_1_STP_PB_LCS;
      AN    "CTRL_SELECTION_CD";
      );
      =     "HYDRAULIC_FUNCTIONS_DB".PUMP_1_STP_PB_LCS;
      A     L 0.0;
      A(;
      A     "PUMP_2_STA_PB_LCS";
      A     "CTRL_SELECTION_CD";
      O;
      A     "WIN_CC_DB".HY_PUMP_2_STA_PB_LCS;
      AN    "CTRL_SELECTION_CD";
      );
      =     "HYDRAULIC_FUNCTIONS_DB".PUMP_2_STA_PB_LCS;
      A     L 0.0;
      A(;
      A     "PUMP_2_STP_PB_LCS";
      A     "CTRL_SELECTION_CD";
      O;
      A     "WIN_CC_DB".HY_PUMP_2_STA_PB_LCS;
      AN    "CTRL_SELECTION_CD";
      );
      =     "HYDRAULIC_FUNCTIONS_DB".PUMP_2_STP_PB_LCS;
      A     L 0.0;
      A(;
      A     "CIR_PUMP_STA_PB_LCS";
      A     "CTRL_SELECTION_CD";
      O;
      A     "WIN_CC_DB".HY_CIR_PUMP_STA_PB_LCS;
      AN    "CTRL_SELECTION_CD";
      );
      =     "HYDRAULIC_FUNCTIONS_DB".CIR_PUMP_STA_PB_LCS;
      A     L 0.0;
      A(;
      A     "CIR_PUMP_STP_PB_LCS";
      A     "CTRL_SELECTION_CD";
      O;
      A     "WIN_CC_DB".HY_CIR_PUMP_STP_PB_LCS;
      AN    "CTRL_SELECTION_CD";
      );
      =     "HYDRAULIC_FUNCTIONS_DB".CIR_PUMP_STP_PB_LCS;
      A     L 0.0;
      A(;
      A     "COLR_FAN_STA_PB_LCS";
      A     "CTRL_SELECTION_CD";
      O;
      A     "WIN_CC_DB".HY_COLR_FAN_STA_PB_LCS;
      AN    "CTRL_SELECTION_CD";
      );
      =     "HYDRAULIC_FUNCTIONS_DB".COLR_FAN_STA_PB_LCS;
      A     L 0.0;
      A(;
      A     "COLR_FAN_STP_PB_LCS";
      A     "CTRL_SELECTION_CD";
      O;
      A     "WIN_CC_DB".HY_COLR_FAN_STP_PB_LCS;
      AN    "CTRL_SELECTION_CD";
      );
      =     "HYDRAULIC_FUNCTIONS_DB".COLR_FAN_STP_PB_LCS;
      A     L 0.0;
      A(;
      A     "EMG_ACCM_STA_PB_LCS";
      A     "CTRL_SELECTION_CD";
      O;
      A     "WIN_CC_DB".EMG_ACCM_STA_PB_LCS;
      AN    "CTRL_SELECTION_CD";
      );
      =     "HYDRAULIC_FUNCTIONS_DB".EMG_ACCM_STA_PB_LCS;
      A     L 0.0;
      A(;
      A     "EMG_ACCM_STP_PB_LCS";
      A     "CTRL_SELECTION_CD";
      O;
      A     "WIN_CC_DB".EMG_ACCM_STP_PB_LCS;
      AN    "CTRL_SELECTION_CD";
      );
      =     "HYDRAULIC_FUNCTIONS_DB".EMG_ACCM_STP_PB_LCS;
      A     L 0.0;
      A     "SHT_OF_VLV_LIN_1_FUL_OPN";
      =     "HYDRAULIC_FUNCTIONS_DB".SHT_OF_VLV_LIN_1_FUL_OPN;
      A     L 0.0;
      A     "SHT_OF_VLV_LIN_2_FUL_OPN";
      =     "HYDRAULIC_FUNCTIONS_DB".SHT_OF_VLV_LIN_2_FUL_OPN;
      A     L 0.0;
      A     "LOW_OIL_TEMP";
      =     "HYDRAULIC_FUNCTIONS_DB".LOW_OIL_TEMP;
      A     L 0.0;
      A     "HIGH_OIL_TEMP";
      =     "HYDRAULIC_FUNCTIONS_DB".HIGH_OIL_TEMP;
      A     L 0.0;
      A     "MAX_OIL_TEMP";
      =     "HYDRAULIC_FUNCTIONS_DB".MAX_OIL_TEMP;
      A     L 0.0;
      A     "LOW_OIL_LEVEL";
      =     "HYDRAULIC_FUNCTIONS_DB".LOW_OIL_LEVEL;
      A     L 0.0;
      A     "MIN_OIL_LEVEL";
      =     "HYDRAULIC_FUNCTIONS_DB".MIN_OIL_LEVEL;
      A     L 0.0;
      A     "RET_LIN_FLTR_CKD";
      =     "HYDRAULIC_FUNCTIONS_DB".RET_LIN_FLTR_CKD;
      A     L 0.0;
      A     "LOW_OIL_PRESS";
      =     "HYDRAULIC_FUNCTIONS_DB".LOW_OIL_PRESS;
      A     L 0.0;
      A     "HIGH_OIL_PRESS";
      =     "HYDRAULIC_FUNCTIONS_DB".HIGH_OIL_PRESS;
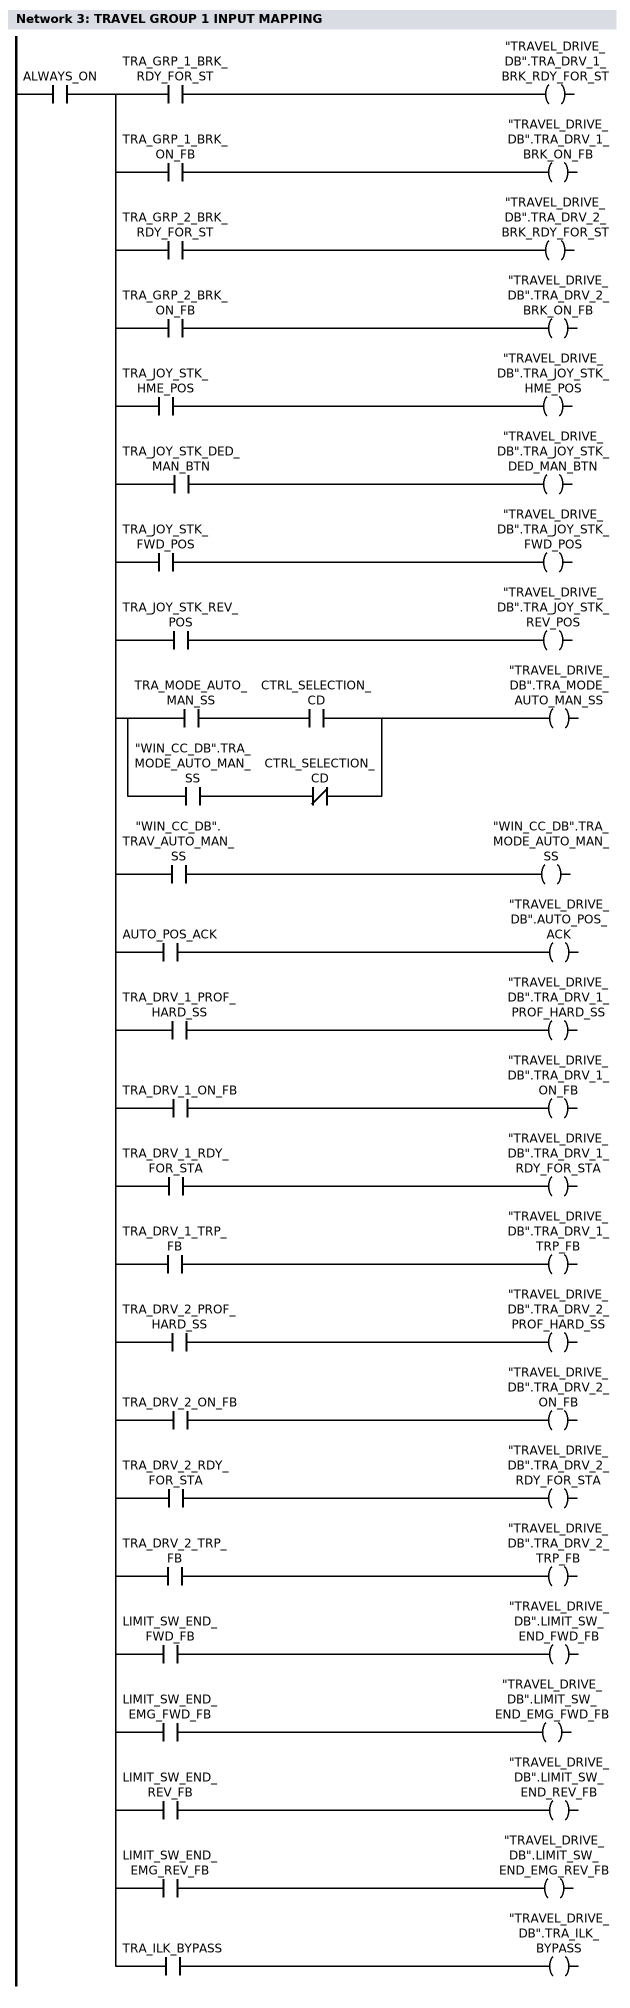
NETWORK
TITLE = TRAVEL GROUP 1 INPUT MAPPING
      A     "ALWAYS_ON";
      =     L 0.0;
      A     L 0.0;
      A     "TRA_GRP_1_BRK_RDY_FOR_ST";
      =     "TRAVEL_DRIVE_DB".TRA_DRV_1_BRK_RDY_FOR_ST;
      A     L 0.0;
      A     "TRA_GRP_1_BRK_ON_FB";
      =     "TRAVEL_DRIVE_DB".TRA_DRV_1_BRK_ON_FB;
      A     L 0.0;
      A     "TRA_GRP_2_BRK_RDY_FOR_ST";
      =     "TRAVEL_DRIVE_DB".TRA_DRV_2_BRK_RDY_FOR_ST;
      A     L 0.0;
      A     "TRA_GRP_2_BRK_ON_FB";
      =     "TRAVEL_DRIVE_DB".TRA_DRV_2_BRK_ON_FB;
      A     L 0.0;
      A     "TRA_JOY_STK_HME_POS";
      =     "TRAVEL_DRIVE_DB".TRA_JOY_STK_HME_POS;
      A     L 0.0;
      A     "TRA_JOY_STK_DED_MAN_BTN";
      =     "TRAVEL_DRIVE_DB".TRA_JOY_STK_DED_MAN_BTN;
      A     L 0.0;
      A     "TRA_JOY_STK_FWD_POS";
      =     "TRAVEL_DRIVE_DB".TRA_JOY_STK_FWD_POS;
      A     L 0.0;
      A     "TRA_JOY_STK_REV_POS";
      =     "TRAVEL_DRIVE_DB".TRA_JOY_STK_REV_POS;
      A     L 0.0;
      A(;
      A     "TRA_MODE_AUTO_MAN_SS";
      A     "CTRL_SELECTION_CD";
      O;
      A     "WIN_CC_DB".TRA_MODE_AUTO_MAN_SS;
      AN    "CTRL_SELECTION_CD";
      );
      =     "TRAVEL_DRIVE_DB".TRA_MODE_AUTO_MAN_SS;
      A     L 0.0;
      A     "WIN_CC_DB".TRAV_AUTO_MAN_SS;
      =     "WIN_CC_DB".TRA_MODE_AUTO_MAN_SS;
      A     L 0.0;
      A     "AUTO_POS_ACK";
      =     "TRAVEL_DRIVE_DB".AUTO_POS_ACK;
      A     L 0.0;
      A     "TRA_DRV_1_PROF_HARD_SS";
      =     "TRAVEL_DRIVE_DB".TRA_DRV_1_PROF_HARD_SS;
      A     L 0.0;
      A     "TRA_DRV_1_ON_FB";
      =     "TRAVEL_DRIVE_DB".TRA_DRV_1_ON_FB;
      A     L 0.0;
      A     "TRA_DRV_1_RDY_FOR_STA";
      =     "TRAVEL_DRIVE_DB".TRA_DRV_1_RDY_FOR_STA;
      A     L 0.0;
      A     "TRA_DRV_1_TRP_FB";
      =     "TRAVEL_DRIVE_DB".TRA_DRV_1_TRP_FB;
      A     L 0.0;
      A     "TRA_DRV_2_PROF_HARD_SS";
      =     "TRAVEL_DRIVE_DB".TRA_DRV_2_PROF_HARD_SS;
      A     L 0.0;
      A     "TRA_DRV_2_ON_FB";
      =     "TRAVEL_DRIVE_DB".TRA_DRV_2_ON_FB;
      A     L 0.0;
      A     "TRA_DRV_2_RDY_FOR_STA";
      =     "TRAVEL_DRIVE_DB".TRA_DRV_2_RDY_FOR_STA;
      A     L 0.0;
      A     "TRA_DRV_2_TRP_FB";
      =     "TRAVEL_DRIVE_DB".TRA_DRV_2_TRP_FB;
      A     L 0.0;
      A     "LIMIT_SW_END_FWD_FB";
      =     "TRAVEL_DRIVE_DB".LIMIT_SW_END_FWD_FB;
      A     L 0.0;
      A     "LIMIT_SW_END_EMG_FWD_FB";
      =     "TRAVEL_DRIVE_DB".LIMIT_SW_END_EMG_FWD_FB;
      A     L 0.0;
      A     "LIMIT_SW_END_REV_FB";
      =     "TRAVEL_DRIVE_DB".LIMIT_SW_END_REV_FB;
      A     L 0.0;
      A     "LIMIT_SW_END_EMG_REV_FB";
      =     "TRAVEL_DRIVE_DB".LIMIT_SW_END_EMG_REV_FB;
      A     L 0.0;
      A     "TRA_ILK_BYPASS";
      =     "TRAVEL_DRIVE_DB".TRA_ILK_BYPASS;
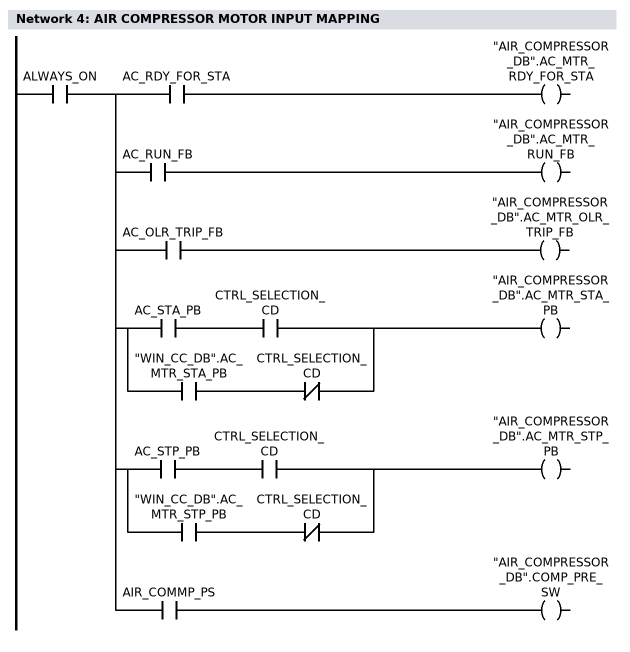
NETWORK
TITLE = AIR COMPRESSOR MOTOR INPUT MAPPING
      A     "ALWAYS_ON";
      =     L 0.0;
      A     L 0.0;
      A     "AC_RDY_FOR_STA";
      =     "AIR_COMPRESSOR_DB".AC_MTR_RDY_FOR_STA;
      A     L 0.0;
      A     "AC_RUN_FB";
      =     "AIR_COMPRESSOR_DB".AC_MTR_RUN_FB;
      A     L 0.0;
      A     "AC_OLR_TRIP_FB";
      =     "AIR_COMPRESSOR_DB".AC_MTR_OLR_TRIP_FB;
      A     L 0.0;
      A(;
      A     "AC_STA_PB";
      A     "CTRL_SELECTION_CD";
      O;
      A     "WIN_CC_DB".AC_MTR_STA_PB;
      AN    "CTRL_SELECTION_CD";
      );
      =     "AIR_COMPRESSOR_DB".AC_MTR_STA_PB;
      A     L 0.0;
      A(;
      A     "AC_STP_PB";
      A     "CTRL_SELECTION_CD";
      O;
      A     "WIN_CC_DB".AC_MTR_STP_PB;
      AN    "CTRL_SELECTION_CD";
      );
      =     "AIR_COMPRESSOR_DB".AC_MTR_STP_PB;
      A     L 0.0;
      A     "AIR_COMMP_PS";
      =     "AIR_COMPRESSOR_DB".COMP_PRE_SW;
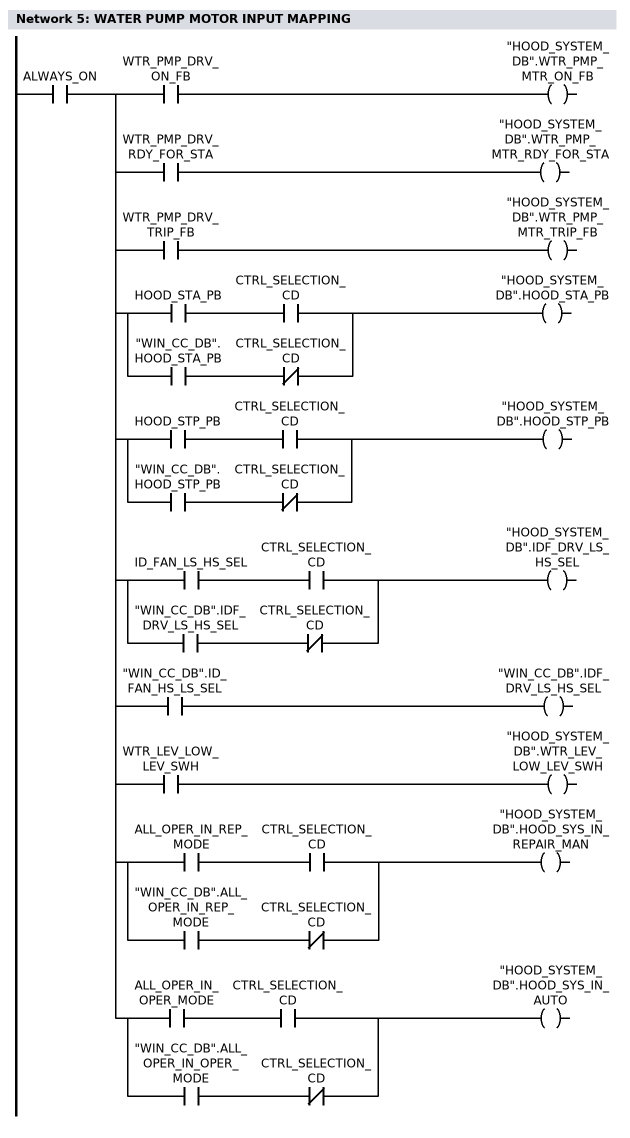
NETWORK
TITLE = WATER PUMP MOTOR INPUT MAPPING
      A     "ALWAYS_ON";
      =     L 0.0;
      A     L 0.0;
      A     "WTR_PMP_DRV_ON_FB";
      =     "HOOD_SYSTEM_DB".WTR_PMP_MTR_ON_FB;
      A     L 0.0;
      A     "WTR_PMP_DRV_RDY_FOR_STA";
      =     "HOOD_SYSTEM_DB".WTR_PMP_MTR_RDY_FOR_STA;
      A     L 0.0;
      A     "WTR_PMP_DRV_TRIP_FB";
      =     "HOOD_SYSTEM_DB".WTR_PMP_MTR_TRIP_FB;
      A     L 0.0;
      A(;
      A     "HOOD_STA_PB";
      A     "CTRL_SELECTION_CD";
      O;
      A     "WIN_CC_DB".HOOD_STA_PB;
      AN    "CTRL_SELECTION_CD";
      );
      =     "HOOD_SYSTEM_DB".HOOD_STA_PB;
      A     L 0.0;
      A(;
      A     "HOOD_STP_PB";
      A     "CTRL_SELECTION_CD";
      O;
      A     "WIN_CC_DB".HOOD_STP_PB;
      AN    "CTRL_SELECTION_CD";
      );
      =     "HOOD_SYSTEM_DB".HOOD_STP_PB;
      A     L 0.0;
      A(;
      A     "ID_FAN_LS_HS_SEL";
      A     "CTRL_SELECTION_CD";
      O;
      A     "WIN_CC_DB".IDF_DRV_LS_HS_SEL;
      AN    "CTRL_SELECTION_CD";
      );
      =     "HOOD_SYSTEM_DB".IDF_DRV_LS_HS_SEL;
      A     L 0.0;
      A     "WIN_CC_DB".ID_FAN_HS_LS_SEL;
      =     "WIN_CC_DB".IDF_DRV_LS_HS_SEL;
      A     L 0.0;
      A     "WTR_LEV_LOW_LEV_SWH";
      =     "HOOD_SYSTEM_DB".WTR_LEV_LOW_LEV_SWH;
      A     L 0.0;
      A(;
      A     "ALL_OPER_IN_REP_MODE";
      A     "CTRL_SELECTION_CD";
      O;
      A     "WIN_CC_DB".ALL_OPER_IN_REP_MODE;
      AN    "CTRL_SELECTION_CD";
      );
      =     "HOOD_SYSTEM_DB".HOOD_SYS_IN_REPAIR_MAN;
      A     L 0.0;
      A(;
      A     "ALL_OPER_IN_OPER_MODE";
      A     "CTRL_SELECTION_CD";
      O;
      A     "WIN_CC_DB".ALL_OPER_IN_OPER_MODE;
      AN    "CTRL_SELECTION_CD";
      );
      =     "HOOD_SYSTEM_DB".HOOD_SYS_IN_AUTO;
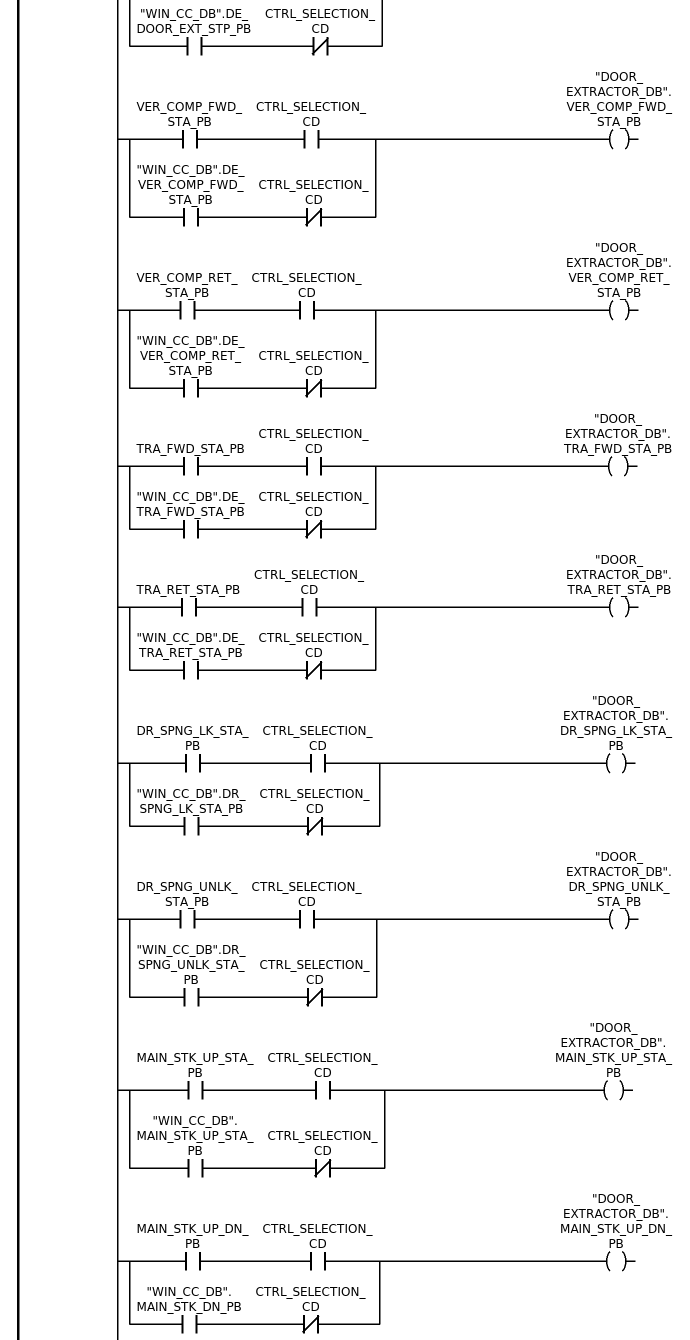
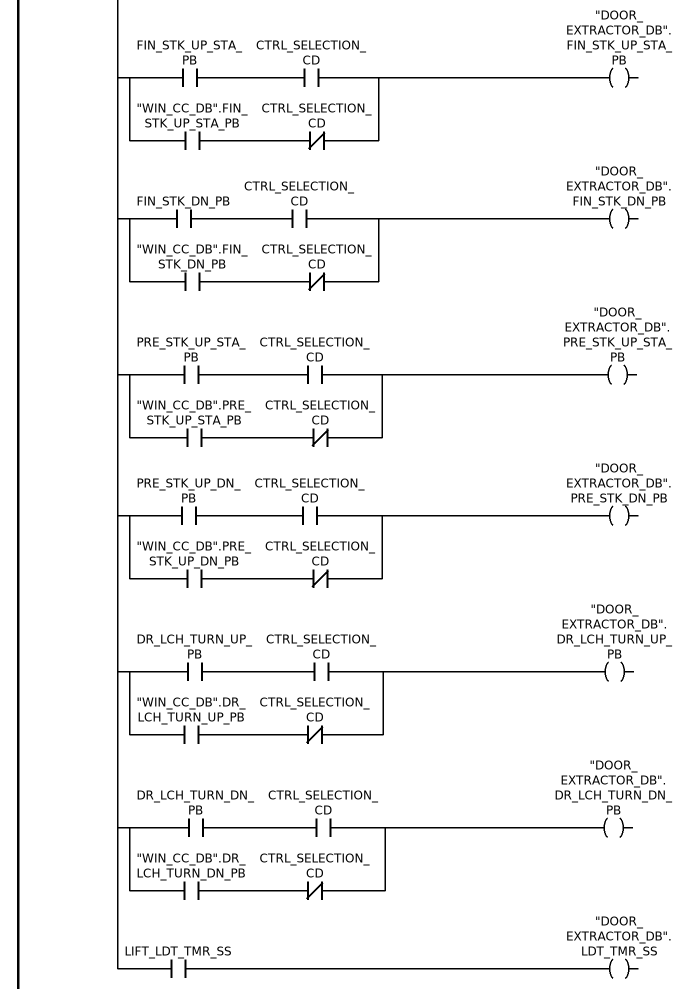
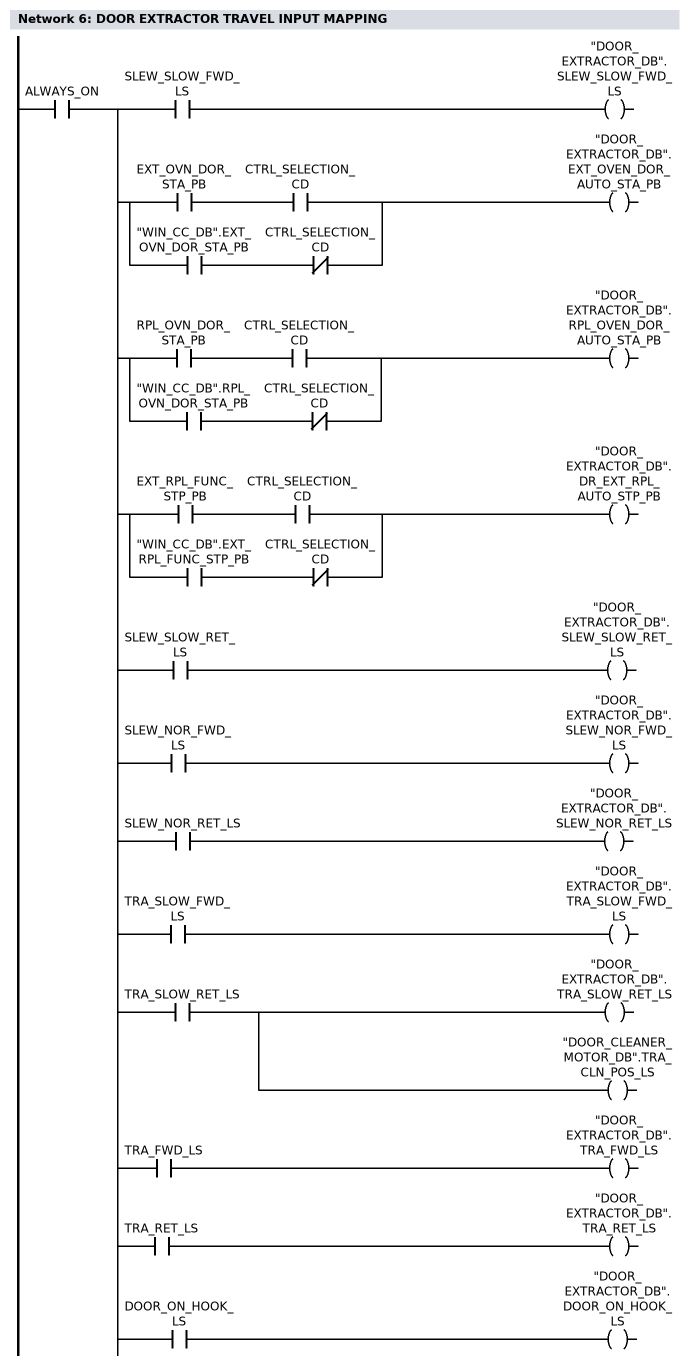
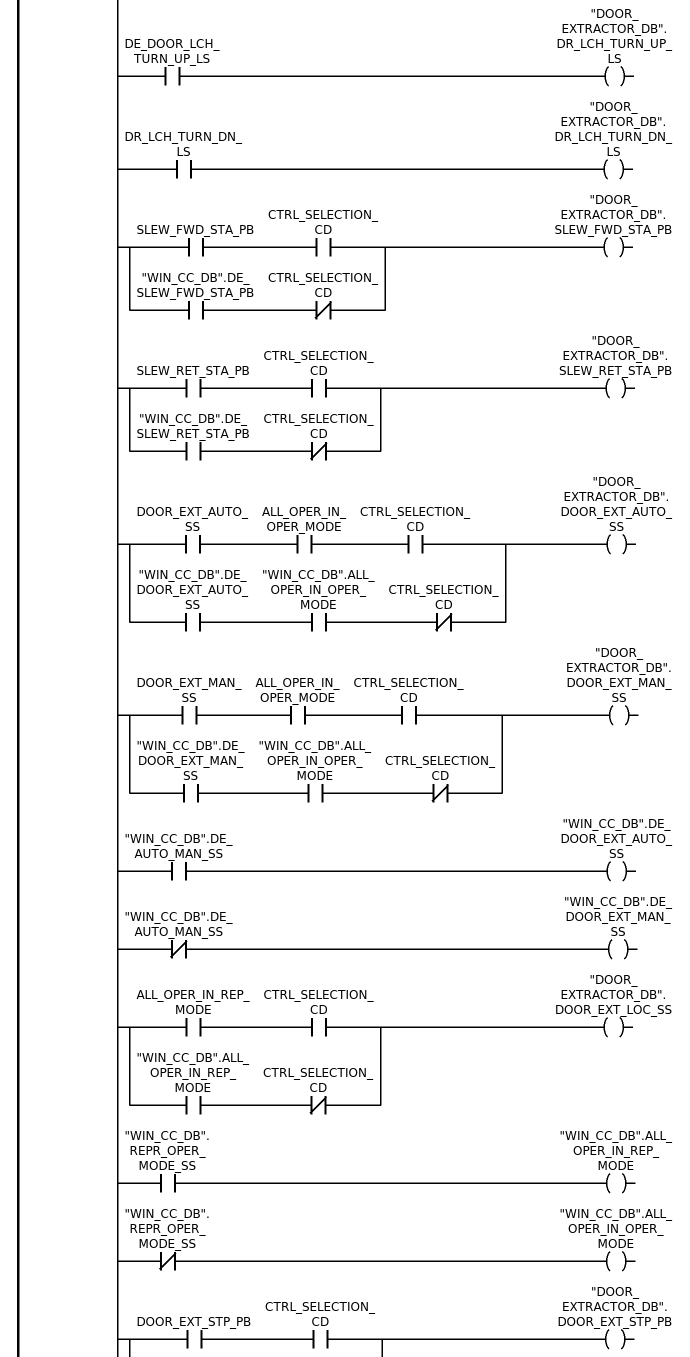
NETWORK
TITLE = DOOR EXTRACTOR TRAVEL INPUT MAPPING
      A     "ALWAYS_ON";
      =     L 0.0;
      A     L 0.0;
      A     "SLEW_SLOW_FWD_LS";
      =     "DOOR_EXTRACTOR_DB".SLEW_SLOW_FWD_LS;
      A     L 0.0;
      A(;
      A     "EXT_OVN_DOR_STA_PB";
      A     "CTRL_SELECTION_CD";
      O;
      A     "WIN_CC_DB".EXT_OVN_DOR_STA_PB;
      AN    "CTRL_SELECTION_CD";
      );
      =     "DOOR_EXTRACTOR_DB".EXT_OVEN_DOR_AUTO_STA_PB;
      A     L 0.0;
      A(;
      A     "RPL_OVN_DOR_STA_PB";
      A     "CTRL_SELECTION_CD";
      O;
      A     "WIN_CC_DB".RPL_OVN_DOR_STA_PB;
      AN    "CTRL_SELECTION_CD";
      );
      =     "DOOR_EXTRACTOR_DB".RPL_OVEN_DOR_AUTO_STA_PB;
      A     L 0.0;
      A(;
      A     "EXT_RPL_FUNC_STP_PB";
      A     "CTRL_SELECTION_CD";
      O;
      A     "WIN_CC_DB".EXT_RPL_FUNC_STP_PB;
      AN    "CTRL_SELECTION_CD";
      );
      =     "DOOR_EXTRACTOR_DB".DR_EXT_RPL_AUTO_STP_PB;
      A     L 0.0;
      A     "SLEW_SLOW_RET_LS";
      =     "DOOR_EXTRACTOR_DB".SLEW_SLOW_RET_LS;
      A     L 0.0;
      A     "SLEW_NOR_FWD_LS";
      =     "DOOR_EXTRACTOR_DB".SLEW_NOR_FWD_LS;
      A     L 0.0;
      A     "SLEW_NOR_RET_LS";
      =     "DOOR_EXTRACTOR_DB".SLEW_NOR_RET_LS;
      A     L 0.0;
      A     "TRA_SLOW_FWD_LS";
      =     "DOOR_EXTRACTOR_DB".TRA_SLOW_FWD_LS;
      A     L 0.0;
      A     "TRA_SLOW_RET_LS";
      =     "DOOR_EXTRACTOR_DB".TRA_SLOW_RET_LS;
      =     "DOOR_CLEANER_MOTOR_DB".TRA_CLN_POS_LS;
      A     L 0.0;
      A     "TRA_FWD_LS";
      =     "DOOR_EXTRACTOR_DB".TRA_FWD_LS;
      A     L 0.0;
      A     "TRA_RET_LS";
      =     "DOOR_EXTRACTOR_DB".TRA_RET_LS;
      A     L 0.0;
      A     "DOOR_ON_HOOK_LS";
      =     "DOOR_EXTRACTOR_DB".DOOR_ON_HOOK_LS;
      A     L 0.0;
      A     "DE_DOOR_LCH_TURN_UP_LS";
      =     "DOOR_EXTRACTOR_DB".DR_LCH_TURN_UP_LS;
      A     L 0.0;
      A     "DR_LCH_TURN_DN_LS";
      =     "DOOR_EXTRACTOR_DB".DR_LCH_TURN_DN_LS;
      A     L 0.0;
      A(;
      A     "SLEW_FWD_STA_PB";
      A     "CTRL_SELECTION_CD";
      O;
      A     "WIN_CC_DB".DE_SLEW_FWD_STA_PB;
      AN    "CTRL_SELECTION_CD";
      );
      =     "DOOR_EXTRACTOR_DB".SLEW_FWD_STA_PB;
      A     L 0.0;
      A(;
      A     "SLEW_RET_STA_PB";
      A     "CTRL_SELECTION_CD";
      O;
      A     "WIN_CC_DB".DE_SLEW_RET_STA_PB;
      AN    "CTRL_SELECTION_CD";
      );
      =     "DOOR_EXTRACTOR_DB".SLEW_RET_STA_PB;
      A     L 0.0;
      A(;
      A     "DOOR_EXT_AUTO_SS";
      A     "ALL_OPER_IN_OPER_MODE";
      A     "CTRL_SELECTION_CD";
      O;
      A     "WIN_CC_DB".DE_DOOR_EXT_AUTO_SS;
      A     "WIN_CC_DB".ALL_OPER_IN_OPER_MODE;
      AN    "CTRL_SELECTION_CD";
      );
      =     "DOOR_EXTRACTOR_DB".DOOR_EXT_AUTO_SS;
      A     L 0.0;
      A(;
      A     "DOOR_EXT_MAN_SS";
      A     "ALL_OPER_IN_OPER_MODE";
      A     "CTRL_SELECTION_CD";
      O;
      A     "WIN_CC_DB".DE_DOOR_EXT_MAN_SS;
      A     "WIN_CC_DB".ALL_OPER_IN_OPER_MODE;
      AN    "CTRL_SELECTION_CD";
      );
      =     "DOOR_EXTRACTOR_DB".DOOR_EXT_MAN_SS;
      A     L 0.0;
      A     "WIN_CC_DB".DE_AUTO_MAN_SS;
      =     "WIN_CC_DB".DE_DOOR_EXT_AUTO_SS;
      A     L 0.0;
      AN    "WIN_CC_DB".DE_AUTO_MAN_SS;
      =     "WIN_CC_DB".DE_DOOR_EXT_MAN_SS;
      A     L 0.0;
      A(;
      A     "ALL_OPER_IN_REP_MODE";
      A     "CTRL_SELECTION_CD";
      O;
      A     "WIN_CC_DB".ALL_OPER_IN_REP_MODE;
      AN    "CTRL_SELECTION_CD";
      );
      =     "DOOR_EXTRACTOR_DB".DOOR_EXT_LOC_SS;
      A     L 0.0;
      A     "WIN_CC_DB".REPR_OPER_MODE_SS;
      =     "WIN_CC_DB".ALL_OPER_IN_REP_MODE;
      A     L 0.0;
      AN    "WIN_CC_DB".REPR_OPER_MODE_SS;
      =     "WIN_CC_DB".ALL_OPER_IN_OPER_MODE;
      A     L 0.0;
      A(;
      A     "DOOR_EXT_STP_PB";
      A     "CTRL_SELECTION_CD";
      O;
      A     "WIN_CC_DB".DE_DOOR_EXT_STP_PB;
      AN    "CTRL_SELECTION_CD";
      );
      =     "DOOR_EXTRACTOR_DB".DOOR_EXT_STP_PB;
      A     L 0.0;
      A(;
      A     "VER_COMP_FWD_STA_PB";
      A     "CTRL_SELECTION_CD";
      O;
      A     "WIN_CC_DB".DE_VER_COMP_FWD_STA_PB;
      AN    "CTRL_SELECTION_CD";
      );
      =     "DOOR_EXTRACTOR_DB".VER_COMP_FWD_STA_PB;
      A     L 0.0;
      A(;
      A     "VER_COMP_RET_STA_PB";
      A     "CTRL_SELECTION_CD";
      O;
      A     "WIN_CC_DB".DE_VER_COMP_RET_STA_PB;
      AN    "CTRL_SELECTION_CD";
      );
      =     "DOOR_EXTRACTOR_DB".VER_COMP_RET_STA_PB;
      A     L 0.0;
      A(;
      A     "TRA_FWD_STA_PB";
      A     "CTRL_SELECTION_CD";
      O;
      A     "WIN_CC_DB".DE_TRA_FWD_STA_PB;
      AN    "CTRL_SELECTION_CD";
      );
      =     "DOOR_EXTRACTOR_DB".TRA_FWD_STA_PB;
      A     L 0.0;
      A(;
      A     "TRA_RET_STA_PB";
      A     "CTRL_SELECTION_CD";
      O;
      A     "WIN_CC_DB".DE_TRA_RET_STA_PB;
      AN    "CTRL_SELECTION_CD";
      );
      =     "DOOR_EXTRACTOR_DB".TRA_RET_STA_PB;
      A     L 0.0;
      A(;
      A     "DR_SPNG_LK_STA_PB";
      A     "CTRL_SELECTION_CD";
      O;
      A     "WIN_CC_DB".DR_SPNG_LK_STA_PB;
      AN    "CTRL_SELECTION_CD";
      );
      =     "DOOR_EXTRACTOR_DB".DR_SPNG_LK_STA_PB;
      A     L 0.0;
      A(;
      A     "DR_SPNG_UNLK_STA_PB";
      A     "CTRL_SELECTION_CD";
      O;
      A     "WIN_CC_DB".DR_SPNG_UNLK_STA_PB;
      AN    "CTRL_SELECTION_CD";
      );
      =     "DOOR_EXTRACTOR_DB".DR_SPNG_UNLK_STA_PB;
      A     L 0.0;
      A(;
      A     "MAIN_STK_UP_STA_PB";
      A     "CTRL_SELECTION_CD";
      O;
      A     "WIN_CC_DB".MAIN_STK_UP_STA_PB;
      AN    "CTRL_SELECTION_CD";
      );
      =     "DOOR_EXTRACTOR_DB".MAIN_STK_UP_STA_PB;
      A     L 0.0;
      A(;
      A     "MAIN_STK_UP_DN_PB";
      A     "CTRL_SELECTION_CD";
      O;
      A     "WIN_CC_DB".MAIN_STK_DN_PB;
      AN    "CTRL_SELECTION_CD";
      );
      =     "DOOR_EXTRACTOR_DB".MAIN_STK_UP_DN_PB;
      A     L 0.0;
      A(;
      A     "FIN_STK_UP_STA_PB";
      A     "CTRL_SELECTION_CD";
      O;
      A     "WIN_CC_DB".FIN_STK_UP_STA_PB;
      AN    "CTRL_SELECTION_CD";
      );
      =     "DOOR_EXTRACTOR_DB".FIN_STK_UP_STA_PB;
      A     L 0.0;
      A(;
      A     "FIN_STK_DN_PB";
      A     "CTRL_SELECTION_CD";
      O;
      A     "WIN_CC_DB".FIN_STK_DN_PB;
      AN    "CTRL_SELECTION_CD";
      );
      =     "DOOR_EXTRACTOR_DB".FIN_STK_DN_PB;
      A     L 0.0;
      A(;
      A     "PRE_STK_UP_STA_PB";
      A     "CTRL_SELECTION_CD";
      O;
      A     "WIN_CC_DB".PRE_STK_UP_STA_PB;
      AN    "CTRL_SELECTION_CD";
      );
      =     "DOOR_EXTRACTOR_DB".PRE_STK_UP_STA_PB;
      A     L 0.0;
      A(;
      A     "PRE_STK_UP_DN_PB";
      A     "CTRL_SELECTION_CD";
      O;
      A     "WIN_CC_DB".PRE_STK_UP_DN_PB;
      AN    "CTRL_SELECTION_CD";
      );
      =     "DOOR_EXTRACTOR_DB".PRE_STK_DN_PB;
      A     L 0.0;
      A(;
      A     "DR_LCH_TURN_UP_PB";
      A     "CTRL_SELECTION_CD";
      O;
      A     "WIN_CC_DB".DR_LCH_TURN_UP_PB;
      AN    "CTRL_SELECTION_CD";
      );
      =     "DOOR_EXTRACTOR_DB".DR_LCH_TURN_UP_PB;
      A     L 0.0;
      A(;
      A     "DR_LCH_TURN_DN_PB";
      A     "CTRL_SELECTION_CD";
      O;
      A     "WIN_CC_DB".DR_LCH_TURN_DN_PB;
      AN    "CTRL_SELECTION_CD";
      );
      =     "DOOR_EXTRACTOR_DB".DR_LCH_TURN_DN_PB;
      A     L 0.0;
      A     "LIFT_LDT_TMR_SS";
      =     "DOOR_EXTRACTOR_DB".LDT_TMR_SS;
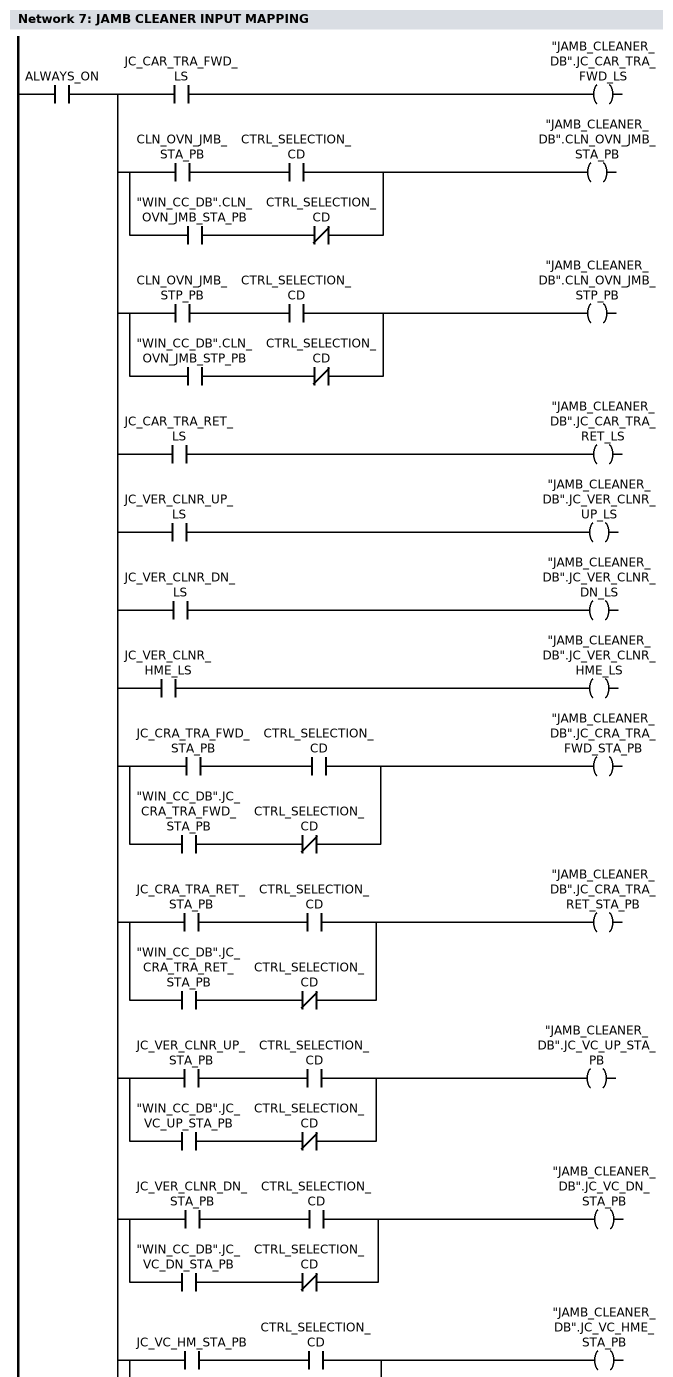
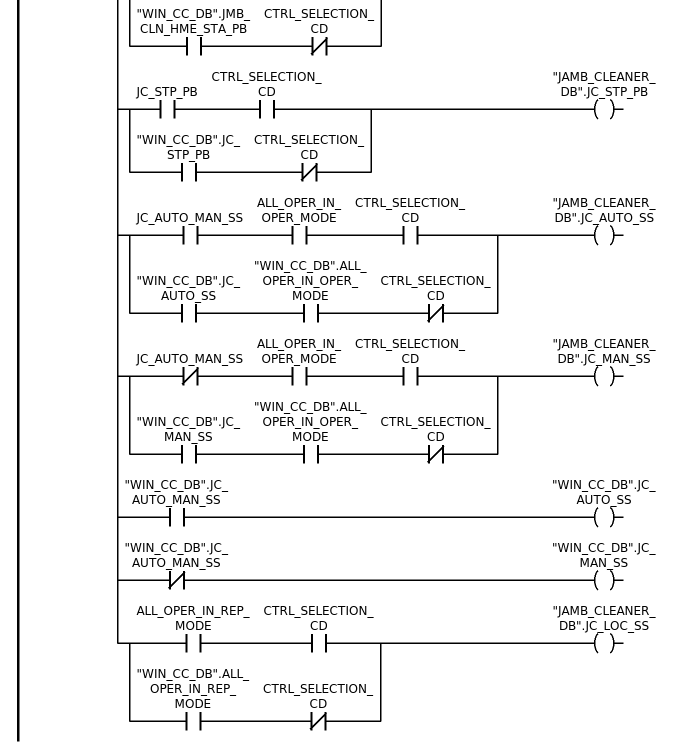
NETWORK
TITLE = JAMB CLEANER INPUT MAPPING
      A     "ALWAYS_ON";
      =     L 0.0;
      A     L 0.0;
      A     "JC_CAR_TRA_FWD_LS";
      =     "JAMB_CLEANER_DB".JC_CAR_TRA_FWD_LS;
      A     L 0.0;
      A(;
      A     "CLN_OVN_JMB_STA_PB";
      A     "CTRL_SELECTION_CD";
      O;
      A     "WIN_CC_DB".CLN_OVN_JMB_STA_PB;
      AN    "CTRL_SELECTION_CD";
      );
      =     "JAMB_CLEANER_DB".CLN_OVN_JMB_STA_PB;
      A     L 0.0;
      A(;
      A     "CLN_OVN_JMB_STP_PB";
      A     "CTRL_SELECTION_CD";
      O;
      A     "WIN_CC_DB".CLN_OVN_JMB_STP_PB;
      AN    "CTRL_SELECTION_CD";
      );
      =     "JAMB_CLEANER_DB".CLN_OVN_JMB_STP_PB;
      A     L 0.0;
      A     "JC_CAR_TRA_RET_LS";
      =     "JAMB_CLEANER_DB".JC_CAR_TRA_RET_LS;
      A     L 0.0;
      A     "JC_VER_CLNR_UP_LS";
      =     "JAMB_CLEANER_DB".JC_VER_CLNR_UP_LS;
      A     L 0.0;
      A     "JC_VER_CLNR_DN_LS";
      =     "JAMB_CLEANER_DB".JC_VER_CLNR_DN_LS;
      A     L 0.0;
      A     "JC_VER_CLNR_HME_LS";
      =     "JAMB_CLEANER_DB".JC_VER_CLNR_HME_LS;
      A     L 0.0;
      A(;
      A     "JC_CRA_TRA_FWD_STA_PB";
      A     "CTRL_SELECTION_CD";
      O;
      A     "WIN_CC_DB".JC_CRA_TRA_FWD_STA_PB;
      AN    "CTRL_SELECTION_CD";
      );
      =     "JAMB_CLEANER_DB".JC_CRA_TRA_FWD_STA_PB;
      A     L 0.0;
      A(;
      A     "JC_CRA_TRA_RET_STA_PB";
      A     "CTRL_SELECTION_CD";
      O;
      A     "WIN_CC_DB".JC_CRA_TRA_RET_STA_PB;
      AN    "CTRL_SELECTION_CD";
      );
      =     "JAMB_CLEANER_DB".JC_CRA_TRA_RET_STA_PB;
      A     L 0.0;
      A(;
      A     "JC_VER_CLNR_UP_STA_PB";
      A     "CTRL_SELECTION_CD";
      O;
      A     "WIN_CC_DB".JC_VC_UP_STA_PB;
      AN    "CTRL_SELECTION_CD";
      );
      =     "JAMB_CLEANER_DB".JC_VC_UP_STA_PB;
      A     L 0.0;
      A(;
      A     "JC_VER_CLNR_DN_STA_PB";
      A     "CTRL_SELECTION_CD";
      O;
      A     "WIN_CC_DB".JC_VC_DN_STA_PB;
      AN    "CTRL_SELECTION_CD";
      );
      =     "JAMB_CLEANER_DB".JC_VC_DN_STA_PB;
      A     L 0.0;
      A(;
      A     "JC_VC_HM_STA_PB";
      A     "CTRL_SELECTION_CD";
      O;
      A     "WIN_CC_DB".JMB_CLN_HME_STA_PB;
      AN    "CTRL_SELECTION_CD";
      );
      =     "JAMB_CLEANER_DB".JC_VC_HME_STA_PB;
      A     L 0.0;
      A(;
      A     "JC_STP_PB";
      A     "CTRL_SELECTION_CD";
      O;
      A     "WIN_CC_DB".JC_STP_PB;
      AN    "CTRL_SELECTION_CD";
      );
      =     "JAMB_CLEANER_DB".JC_STP_PB;
      A     L 0.0;
      A(;
      A     "JC_AUTO_MAN_SS";
      A     "ALL_OPER_IN_OPER_MODE";
      A     "CTRL_SELECTION_CD";
      O;
      A     "WIN_CC_DB".JC_AUTO_SS;
      A     "WIN_CC_DB".ALL_OPER_IN_OPER_MODE;
      AN    "CTRL_SELECTION_CD";
      );
      =     "JAMB_CLEANER_DB".JC_AUTO_SS;
      A     L 0.0;
      A(;
      AN    "JC_AUTO_MAN_SS";
      A     "ALL_OPER_IN_OPER_MODE";
      A     "CTRL_SELECTION_CD";
      O;
      A     "WIN_CC_DB".JC_MAN_SS;
      A     "WIN_CC_DB".ALL_OPER_IN_OPER_MODE;
      AN    "CTRL_SELECTION_CD";
      );
      =     "JAMB_CLEANER_DB".JC_MAN_SS;
      A     L 0.0;
      A     "WIN_CC_DB".JC_AUTO_MAN_SS;
      =     "WIN_CC_DB".JC_AUTO_SS;
      A     L 0.0;
      AN    "WIN_CC_DB".JC_AUTO_MAN_SS;
      =     "WIN_CC_DB".JC_MAN_SS;
      A     L 0.0;
      A(;
      A     "ALL_OPER_IN_REP_MODE";
      A     "CTRL_SELECTION_CD";
      O;
      A     "WIN_CC_DB".ALL_OPER_IN_REP_MODE;
      AN    "CTRL_SELECTION_CD";
      );
      =     "JAMB_CLEANER_DB".JC_LOC_SS;
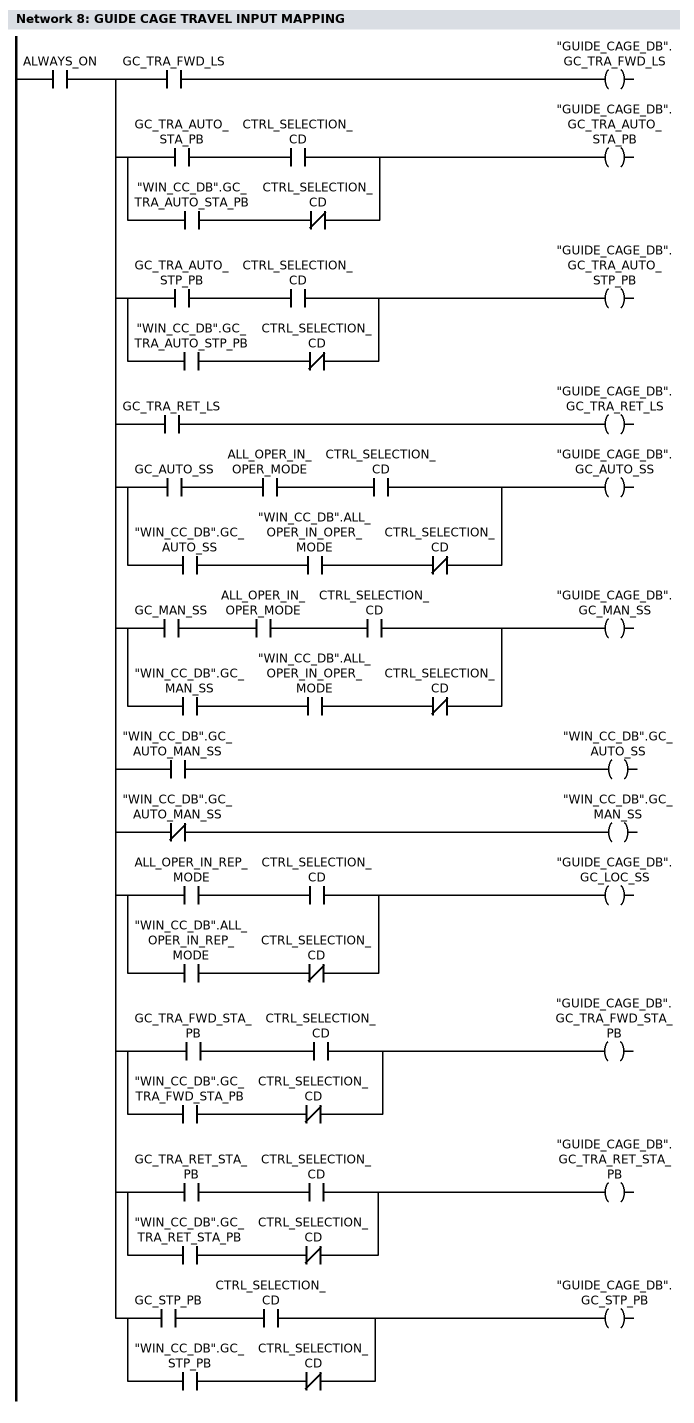
NETWORK
TITLE = GUIDE CAGE TRAVEL INPUT MAPPING
      A     "ALWAYS_ON";
      =     L 0.0;
      A     L 0.0;
      A     "GC_TRA_FWD_LS";
      =     "GUIDE_CAGE_DB".GC_TRA_FWD_LS;
      A     L 0.0;
      A(;
      A     "GC_TRA_AUTO_STA_PB";
      A     "CTRL_SELECTION_CD";
      O;
      A     "WIN_CC_DB".GC_TRA_AUTO_STA_PB;
      AN    "CTRL_SELECTION_CD";
      );
      =     "GUIDE_CAGE_DB".GC_TRA_AUTO_STA_PB;
      A     L 0.0;
      A(;
      A     "GC_TRA_AUTO_STP_PB";
      A     "CTRL_SELECTION_CD";
      O;
      A     "WIN_CC_DB".GC_TRA_AUTO_STP_PB;
      AN    "CTRL_SELECTION_CD";
      );
      =     "GUIDE_CAGE_DB".GC_TRA_AUTO_STP_PB;
      A     L 0.0;
      A     "GC_TRA_RET_LS";
      =     "GUIDE_CAGE_DB".GC_TRA_RET_LS;
      A     L 0.0;
      A(;
      A     "GC_AUTO_SS";
      A     "ALL_OPER_IN_OPER_MODE";
      A     "CTRL_SELECTION_CD";
      O;
      A     "WIN_CC_DB".GC_AUTO_SS;
      A     "WIN_CC_DB".ALL_OPER_IN_OPER_MODE;
      AN    "CTRL_SELECTION_CD";
      );
      =     "GUIDE_CAGE_DB".GC_AUTO_SS;
      A     L 0.0;
      A(;
      A     "GC_MAN_SS";
      A     "ALL_OPER_IN_OPER_MODE";
      A     "CTRL_SELECTION_CD";
      O;
      A     "WIN_CC_DB".GC_MAN_SS;
      A     "WIN_CC_DB".ALL_OPER_IN_OPER_MODE;
      AN    "CTRL_SELECTION_CD";
      );
      =     "GUIDE_CAGE_DB".GC_MAN_SS;
      A     L 0.0;
      A     "WIN_CC_DB".GC_AUTO_MAN_SS;
      =     "WIN_CC_DB".GC_AUTO_SS;
      A     L 0.0;
      AN    "WIN_CC_DB".GC_AUTO_MAN_SS;
      =     "WIN_CC_DB".GC_MAN_SS;
      A     L 0.0;
      A(;
      A     "ALL_OPER_IN_REP_MODE";
      A     "CTRL_SELECTION_CD";
      O;
      A     "WIN_CC_DB".ALL_OPER_IN_REP_MODE;
      AN    "CTRL_SELECTION_CD";
      );
      =     "GUIDE_CAGE_DB".GC_LOC_SS;
      A     L 0.0;
      A(;
      A     "GC_TRA_FWD_STA_PB";
      A     "CTRL_SELECTION_CD";
      O;
      A     "WIN_CC_DB".GC_TRA_FWD_STA_PB;
      AN    "CTRL_SELECTION_CD";
      );
      =     "GUIDE_CAGE_DB".GC_TRA_FWD_STA_PB;
      A     L 0.0;
      A(;
      A     "GC_TRA_RET_STA_PB";
      A     "CTRL_SELECTION_CD";
      O;
      A     "WIN_CC_DB".GC_TRA_RET_STA_PB;
      AN    "CTRL_SELECTION_CD";
      );
      =     "GUIDE_CAGE_DB".GC_TRA_RET_STA_PB;
      A     L 0.0;
      A(;
      A     "GC_STP_PB";
      A     "CTRL_SELECTION_CD";
      O;
      A     "WIN_CC_DB".GC_STP_PB;
      AN    "CTRL_SELECTION_CD";
      );
      =     "GUIDE_CAGE_DB".GC_STP_PB;
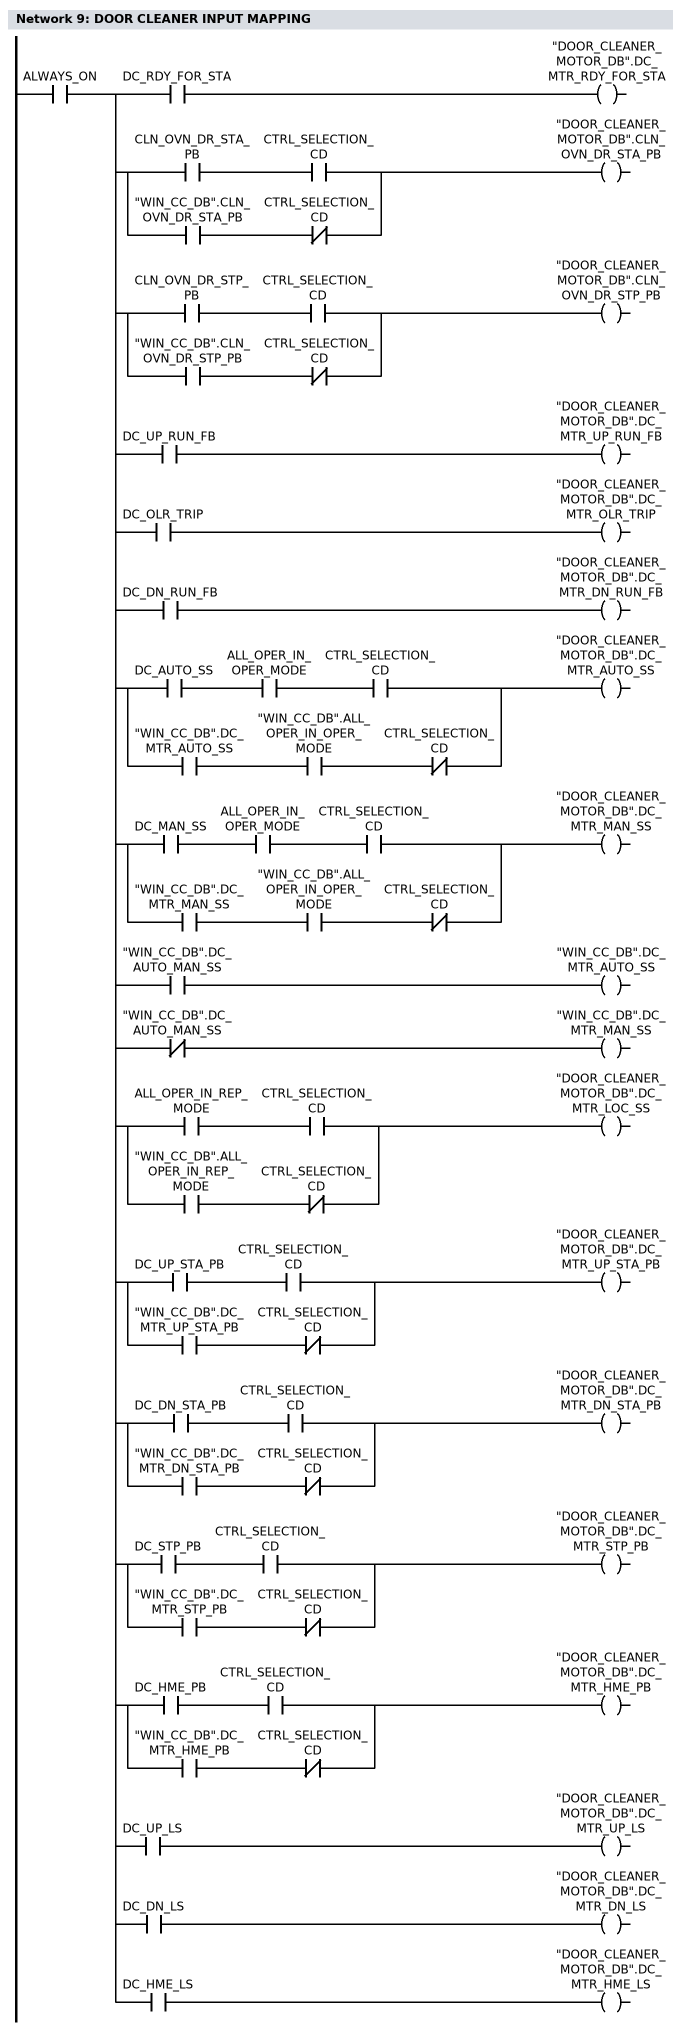
NETWORK
TITLE = DOOR CLEANER INPUT MAPPING
      A     "ALWAYS_ON";
      =     L 0.0;
      A     L 0.0;
      A     "DC_RDY_FOR_STA";
      =     "DOOR_CLEANER_MOTOR_DB".DC_MTR_RDY_FOR_STA;
      A     L 0.0;
      A(;
      A     "CLN_OVN_DR_STA_PB";
      A     "CTRL_SELECTION_CD";
      O;
      A     "WIN_CC_DB".CLN_OVN_DR_STA_PB;
      AN    "CTRL_SELECTION_CD";
      );
      =     "DOOR_CLEANER_MOTOR_DB".CLN_OVN_DR_STA_PB;
      A     L 0.0;
      A(;
      A     "CLN_OVN_DR_STP_PB";
      A     "CTRL_SELECTION_CD";
      O;
      A     "WIN_CC_DB".CLN_OVN_DR_STP_PB;
      AN    "CTRL_SELECTION_CD";
      );
      =     "DOOR_CLEANER_MOTOR_DB".CLN_OVN_DR_STP_PB;
      A     L 0.0;
      A     "DC_UP_RUN_FB";
      =     "DOOR_CLEANER_MOTOR_DB".DC_MTR_UP_RUN_FB;
      A     L 0.0;
      A     "DC_OLR_TRIP";
      =     "DOOR_CLEANER_MOTOR_DB".DC_MTR_OLR_TRIP;
      A     L 0.0;
      A     "DC_DN_RUN_FB";
      =     "DOOR_CLEANER_MOTOR_DB".DC_MTR_DN_RUN_FB;
      A     L 0.0;
      A(;
      A     "DC_AUTO_SS";
      A     "ALL_OPER_IN_OPER_MODE";
      A     "CTRL_SELECTION_CD";
      O;
      A     "WIN_CC_DB".DC_MTR_AUTO_SS;
      A     "WIN_CC_DB".ALL_OPER_IN_OPER_MODE;
      AN    "CTRL_SELECTION_CD";
      );
      =     "DOOR_CLEANER_MOTOR_DB".DC_MTR_AUTO_SS;
      A     L 0.0;
      A(;
      A     "DC_MAN_SS";
      A     "ALL_OPER_IN_OPER_MODE";
      A     "CTRL_SELECTION_CD";
      O;
      A     "WIN_CC_DB".DC_MTR_MAN_SS;
      A     "WIN_CC_DB".ALL_OPER_IN_OPER_MODE;
      AN    "CTRL_SELECTION_CD";
      );
      =     "DOOR_CLEANER_MOTOR_DB".DC_MTR_MAN_SS;
      A     L 0.0;
      A     "WIN_CC_DB".DC_AUTO_MAN_SS;
      =     "WIN_CC_DB".DC_MTR_AUTO_SS;
      A     L 0.0;
      AN    "WIN_CC_DB".DC_AUTO_MAN_SS;
      =     "WIN_CC_DB".DC_MTR_MAN_SS;
      A     L 0.0;
      A(;
      A     "ALL_OPER_IN_REP_MODE";
      A     "CTRL_SELECTION_CD";
      O;
      A     "WIN_CC_DB".ALL_OPER_IN_REP_MODE;
      AN    "CTRL_SELECTION_CD";
      );
      =     "DOOR_CLEANER_MOTOR_DB".DC_MTR_LOC_SS;
      A     L 0.0;
      A(;
      A     "DC_UP_STA_PB";
      A     "CTRL_SELECTION_CD";
      O;
      A     "WIN_CC_DB".DC_MTR_UP_STA_PB;
      AN    "CTRL_SELECTION_CD";
      );
      =     "DOOR_CLEANER_MOTOR_DB".DC_MTR_UP_STA_PB;
      A     L 0.0;
      A(;
      A     "DC_DN_STA_PB";
      A     "CTRL_SELECTION_CD";
      O;
      A     "WIN_CC_DB".DC_MTR_DN_STA_PB;
      AN    "CTRL_SELECTION_CD";
      );
      =     "DOOR_CLEANER_MOTOR_DB".DC_MTR_DN_STA_PB;
      A     L 0.0;
      A(;
      A     "DC_STP_PB";
      A     "CTRL_SELECTION_CD";
      O;
      A     "WIN_CC_DB".DC_MTR_STP_PB;
      AN    "CTRL_SELECTION_CD";
      );
      =     "DOOR_CLEANER_MOTOR_DB".DC_MTR_STP_PB;
      A     L 0.0;
      A(;
      A     "DC_HME_PB";
      A     "CTRL_SELECTION_CD";
      O;
      A     "WIN_CC_DB".DC_MTR_HME_PB;
      AN    "CTRL_SELECTION_CD";
      );
      =     "DOOR_CLEANER_MOTOR_DB".DC_MTR_HME_PB;
      A     L 0.0;
      A     "DC_UP_LS";
      =     "DOOR_CLEANER_MOTOR_DB".DC_MTR_UP_LS;
      A     L 0.0;
      A     "DC_DN_LS";
      =     "DOOR_CLEANER_MOTOR_DB".DC_MTR_DN_LS;
      A     L 0.0;
      A     "DC_HME_LS";
      =     "DOOR_CLEANER_MOTOR_DB".DC_MTR_HME_LS;
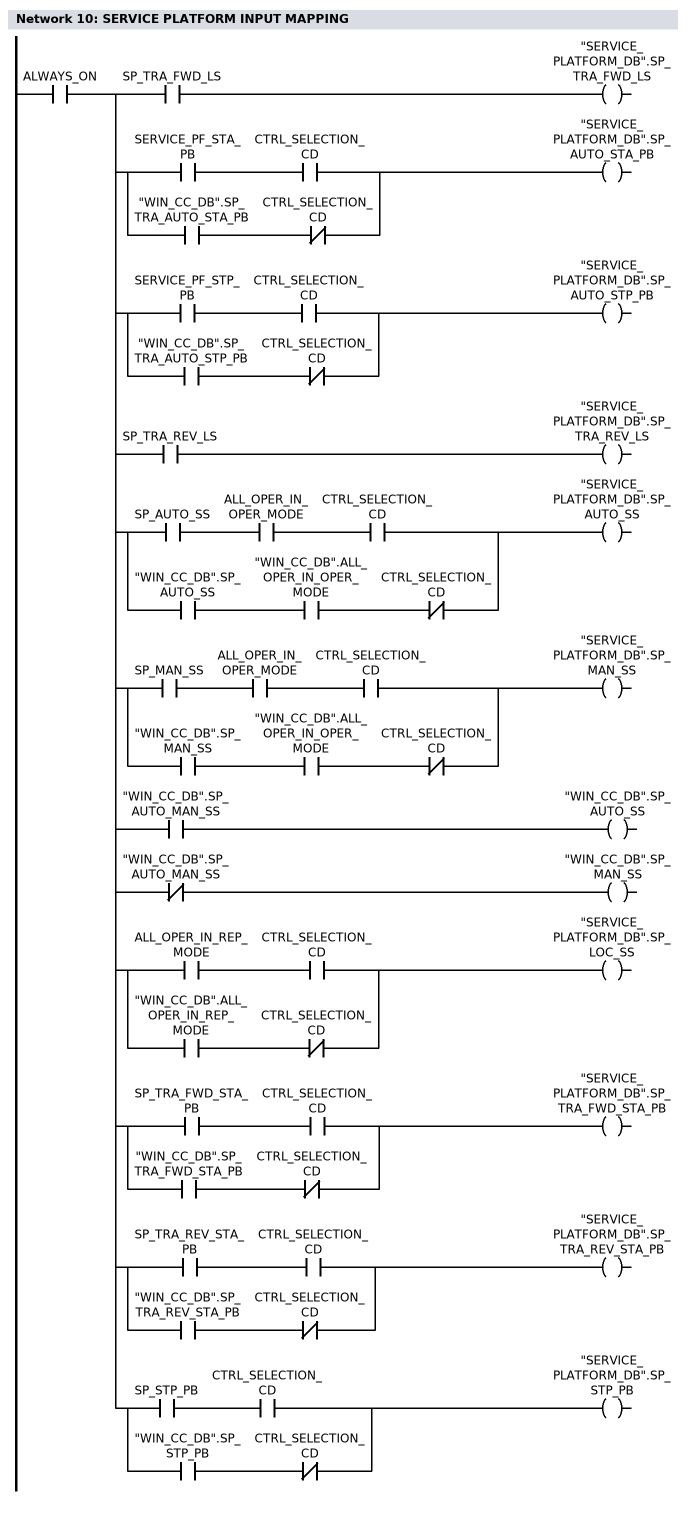
NETWORK
TITLE = SERVICE PLATFORM INPUT MAPPING
      A     "ALWAYS_ON";
      =     L 0.0;
      A     L 0.0;
      A     "SP_TRA_FWD_LS";
      =     "SERVICE_PLATFORM_DB".SP_TRA_FWD_LS;
      A     L 0.0;
      A(;
      A     "SERVICE_PF_STA_PB";
      A     "CTRL_SELECTION_CD";
      O;
      A     "WIN_CC_DB".SP_TRA_AUTO_STA_PB;
      AN    "CTRL_SELECTION_CD";
      );
      =     "SERVICE_PLATFORM_DB".SP_AUTO_STA_PB;
      A     L 0.0;
      A(;
      A     "SERVICE_PF_STP_PB";
      A     "CTRL_SELECTION_CD";
      O;
      A     "WIN_CC_DB".SP_TRA_AUTO_STP_PB;
      AN    "CTRL_SELECTION_CD";
      );
      =     "SERVICE_PLATFORM_DB".SP_AUTO_STP_PB;
      A     L 0.0;
      A     "SP_TRA_REV_LS";
      =     "SERVICE_PLATFORM_DB".SP_TRA_REV_LS;
      A     L 0.0;
      A(;
      A     "SP_AUTO_SS";
      A     "ALL_OPER_IN_OPER_MODE";
      A     "CTRL_SELECTION_CD";
      O;
      A     "WIN_CC_DB".SP_AUTO_SS;
      A     "WIN_CC_DB".ALL_OPER_IN_OPER_MODE;
      AN    "CTRL_SELECTION_CD";
      );
      =     "SERVICE_PLATFORM_DB".SP_AUTO_SS;
      A     L 0.0;
      A(;
      A     "SP_MAN_SS";
      A     "ALL_OPER_IN_OPER_MODE";
      A     "CTRL_SELECTION_CD";
      O;
      A     "WIN_CC_DB".SP_MAN_SS;
      A     "WIN_CC_DB".ALL_OPER_IN_OPER_MODE;
      AN    "CTRL_SELECTION_CD";
      );
      =     "SERVICE_PLATFORM_DB".SP_MAN_SS;
      A     L 0.0;
      A     "WIN_CC_DB".SP_AUTO_MAN_SS;
      =     "WIN_CC_DB".SP_AUTO_SS;
      A     L 0.0;
      AN    "WIN_CC_DB".SP_AUTO_MAN_SS;
      =     "WIN_CC_DB".SP_MAN_SS;
      A     L 0.0;
      A(;
      A     "ALL_OPER_IN_REP_MODE";
      A     "CTRL_SELECTION_CD";
      O;
      A     "WIN_CC_DB".ALL_OPER_IN_REP_MODE;
      AN    "CTRL_SELECTION_CD";
      );
      =     "SERVICE_PLATFORM_DB".SP_LOC_SS;
      A     L 0.0;
      A(;
      A     "SP_TRA_FWD_STA_PB";
      A     "CTRL_SELECTION_CD";
      O;
      A     "WIN_CC_DB".SP_TRA_FWD_STA_PB;
      AN    "CTRL_SELECTION_CD";
      );
      =     "SERVICE_PLATFORM_DB".SP_TRA_FWD_STA_PB;
      A     L 0.0;
      A(;
      A     "SP_TRA_REV_STA_PB";
      A     "CTRL_SELECTION_CD";
      O;
      A     "WIN_CC_DB".SP_TRA_REV_STA_PB;
      AN    "CTRL_SELECTION_CD";
      );
      =     "SERVICE_PLATFORM_DB".SP_TRA_REV_STA_PB;
      A     L 0.0;
      A(;
      A     "SP_STP_PB";
      A     "CTRL_SELECTION_CD";
      O;
      A     "WIN_CC_DB".SP_STP_PB;
      AN    "CTRL_SELECTION_CD";
      );
      =     "SERVICE_PLATFORM_DB".SP_STP_PB;
END_FUNCTION

FUNCTION "OUTPUT_MAPPING" : VOID	// FC 2
AUTHOR : Kamillas
VERSION : 0.1
BEGIN
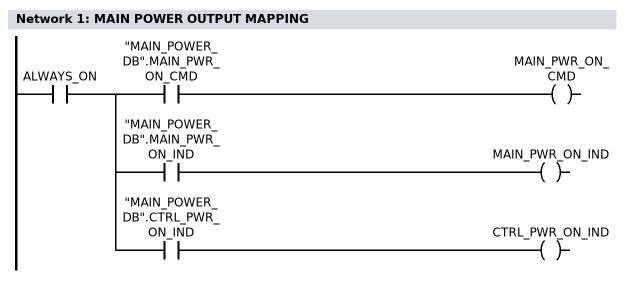
NETWORK
TITLE = MAIN POWER OUTPUT MAPPING
      A     "ALWAYS_ON";
      =     L 0.0;
      A     L 0.0;
      A     "MAIN_POWER_DB".MAIN_PWR_ON_CMD;
      =     "MAIN_PWR_ON_CMD";
      A     L 0.0;
      A     "MAIN_POWER_DB".MAIN_PWR_ON_IND;
      =     "MAIN_PWR_ON_IND";
      A     L 0.0;
      A     "MAIN_POWER_DB".CTRL_PWR_ON_IND;
      =     "CTRL_PWR_ON_IND";
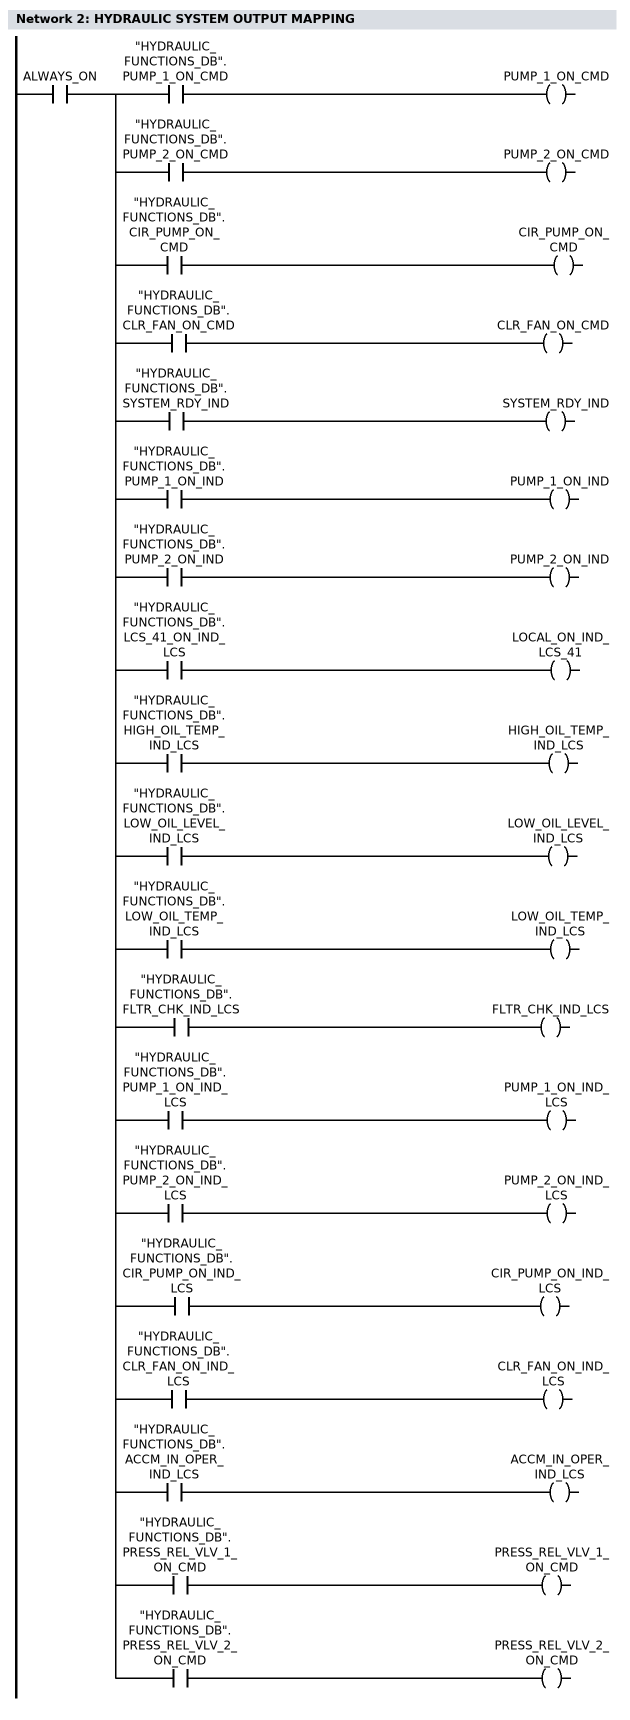
NETWORK
TITLE = HYDRAULIC SYSTEM OUTPUT MAPPING
      A     "ALWAYS_ON";
      =     L 0.0;
      A     L 0.0;
      A     "HYDRAULIC_FUNCTIONS_DB".PUMP_1_ON_CMD;
      =     "PUMP_1_ON_CMD";
      A     L 0.0;
      A     "HYDRAULIC_FUNCTIONS_DB".PUMP_2_ON_CMD;
      =     "PUMP_2_ON_CMD";
      A     L 0.0;
      A     "HYDRAULIC_FUNCTIONS_DB".CIR_PUMP_ON_CMD;
      =     "CIR_PUMP_ON_CMD";
      A     L 0.0;
      A     "HYDRAULIC_FUNCTIONS_DB".CLR_FAN_ON_CMD;
      =     "CLR_FAN_ON_CMD";
      A     L 0.0;
      A     "HYDRAULIC_FUNCTIONS_DB".SYSTEM_RDY_IND;
      =     "SYSTEM_RDY_IND";
      A     L 0.0;
      A     "HYDRAULIC_FUNCTIONS_DB".PUMP_1_ON_IND;
      =     "PUMP_1_ON_IND";
      A     L 0.0;
      A     "HYDRAULIC_FUNCTIONS_DB".PUMP_2_ON_IND;
      =     "PUMP_2_ON_IND";
      A     L 0.0;
      A     "HYDRAULIC_FUNCTIONS_DB".LCS_41_ON_IND_LCS;
      =     "LOCAL_ON_IND_LCS_41";
      A     L 0.0;
      A     "HYDRAULIC_FUNCTIONS_DB".HIGH_OIL_TEMP_IND_LCS;
      =     "HIGH_OIL_TEMP_IND_LCS";
      A     L 0.0;
      A     "HYDRAULIC_FUNCTIONS_DB".LOW_OIL_LEVEL_IND_LCS;
      =     "LOW_OIL_LEVEL_IND_LCS";
      A     L 0.0;
      A     "HYDRAULIC_FUNCTIONS_DB".LOW_OIL_TEMP_IND_LCS;
      =     "LOW_OIL_TEMP_IND_LCS";
      A     L 0.0;
      A     "HYDRAULIC_FUNCTIONS_DB".FLTR_CHK_IND_LCS;
      =     "FLTR_CHK_IND_LCS";
      A     L 0.0;
      A     "HYDRAULIC_FUNCTIONS_DB".PUMP_1_ON_IND_LCS;
      =     "PUMP_1_ON_IND_LCS";
      A     L 0.0;
      A     "HYDRAULIC_FUNCTIONS_DB".PUMP_2_ON_IND_LCS;
      =     "PUMP_2_ON_IND_LCS";
      A     L 0.0;
      A     "HYDRAULIC_FUNCTIONS_DB".CIR_PUMP_ON_IND_LCS;
      =     "CIR_PUMP_ON_IND_LCS";
      A     L 0.0;
      A     "HYDRAULIC_FUNCTIONS_DB".CLR_FAN_ON_IND_LCS;
      =     "CLR_FAN_ON_IND_LCS";
      A     L 0.0;
      A     "HYDRAULIC_FUNCTIONS_DB".ACCM_IN_OPER_IND_LCS;
      =     "ACCM_IN_OPER_IND_LCS";
      A     L 0.0;
      A     "HYDRAULIC_FUNCTIONS_DB".PRESS_REL_VLV_1_ON_CMD;
      =     "PRESS_REL_VLV_1_ON_CMD";
      A     L 0.0;
      A     "HYDRAULIC_FUNCTIONS_DB".PRESS_REL_VLV_2_ON_CMD;
      =     "PRESS_REL_VLV_2_ON_CMD";
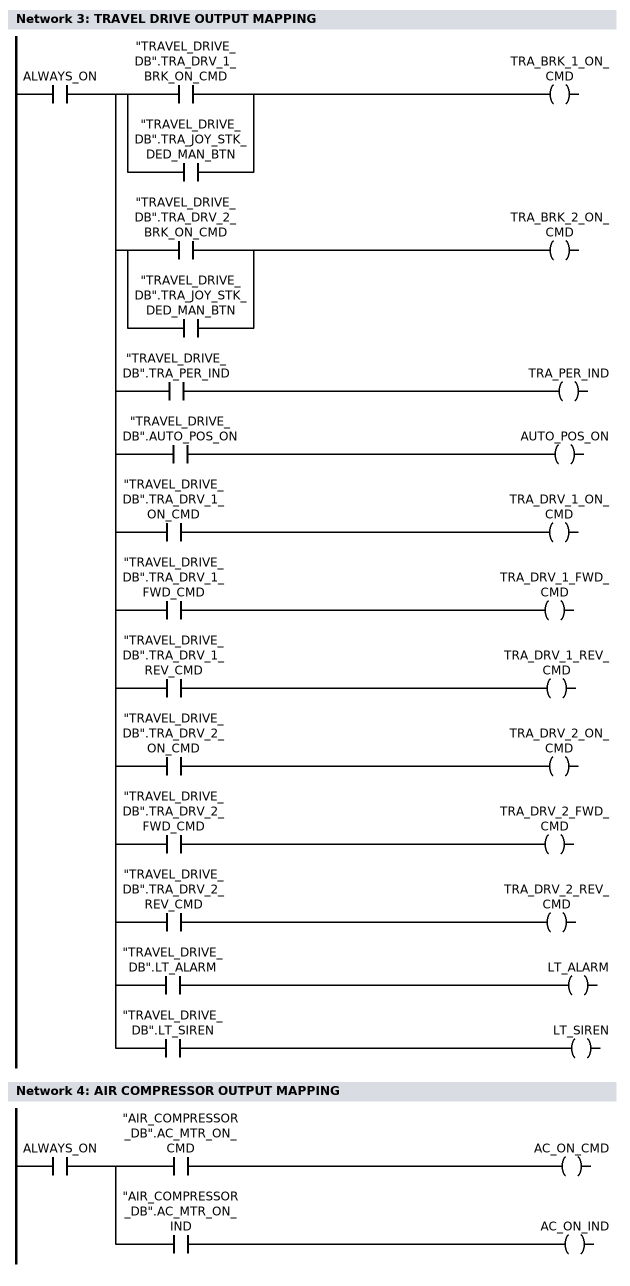
NETWORK
TITLE = TRAVEL DRIVE OUTPUT MAPPING
      A     "ALWAYS_ON";
      =     L 0.0;
      A     L 0.0;
      A(;
      O     "TRAVEL_DRIVE_DB".TRA_DRV_1_BRK_ON_CMD;
      O     "TRAVEL_DRIVE_DB".TRA_JOY_STK_DED_MAN_BTN;
      );
      =     "TRA_BRK_1_ON_CMD";
      A     L 0.0;
      A(;
      O     "TRAVEL_DRIVE_DB".TRA_DRV_2_BRK_ON_CMD;
      O     "TRAVEL_DRIVE_DB".TRA_JOY_STK_DED_MAN_BTN;
      );
      =     "TRA_BRK_2_ON_CMD";
      A     L 0.0;
      A     "TRAVEL_DRIVE_DB".TRA_PER_IND;
      =     "TRA_PER_IND";
      A     L 0.0;
      A     "TRAVEL_DRIVE_DB".AUTO_POS_ON;
      =     "AUTO_POS_ON";
      A     L 0.0;
      A     "TRAVEL_DRIVE_DB".TRA_DRV_1_ON_CMD;
      =     "TRA_DRV_1_ON_CMD";
      A     L 0.0;
      A     "TRAVEL_DRIVE_DB".TRA_DRV_1_FWD_CMD;
      =     "TRA_DRV_1_FWD_CMD";
      A     L 0.0;
      A     "TRAVEL_DRIVE_DB".TRA_DRV_1_REV_CMD;
      =     "TRA_DRV_1_REV_CMD";
      A     L 0.0;
      A     "TRAVEL_DRIVE_DB".TRA_DRV_2_ON_CMD;
      =     "TRA_DRV_2_ON_CMD";
      A     L 0.0;
      A     "TRAVEL_DRIVE_DB".TRA_DRV_2_FWD_CMD;
      =     "TRA_DRV_2_FWD_CMD";
      A     L 0.0;
      A     "TRAVEL_DRIVE_DB".TRA_DRV_2_REV_CMD;
      =     "TRA_DRV_2_REV_CMD";
      A     L 0.0;
      A     "TRAVEL_DRIVE_DB".LT_ALARM;
      =     "LT_ALARM";
      A     L 0.0;
      A     "TRAVEL_DRIVE_DB".LT_SIREN;
      =     "LT_SIREN";
NETWORK
TITLE = AIR COMPRESSOR OUTPUT MAPPING
      A     "ALWAYS_ON";
      =     L 0.0;
      A     L 0.0;
      A     "AIR_COMPRESSOR_DB".AC_MTR_ON_CMD;
      =     "AC_ON_CMD";
      A     L 0.0;
      A     "AIR_COMPRESSOR_DB".AC_MTR_ON_IND;
      =     "AC_ON_IND";
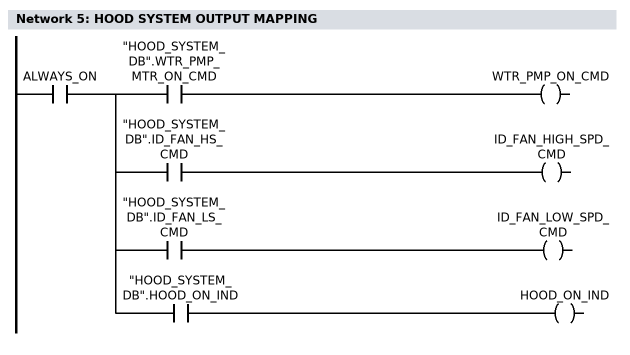
NETWORK
TITLE = HOOD SYSTEM OUTPUT MAPPING
      A     "ALWAYS_ON";
      =     L 0.0;
      A     L 0.0;
      A     "HOOD_SYSTEM_DB".WTR_PMP_MTR_ON_CMD;
      =     "WTR_PMP_ON_CMD";
      A     L 0.0;
      A     "HOOD_SYSTEM_DB".ID_FAN_HS_CMD;
      =     "ID_FAN_HIGH_SPD_CMD";
      A     L 0.0;
      A     "HOOD_SYSTEM_DB".ID_FAN_LS_CMD;
      =     "ID_FAN_LOW_SPD_CMD";
      A     L 0.0;
      A     "HOOD_SYSTEM_DB".HOOD_ON_IND;
      =     "HOOD_ON_IND";
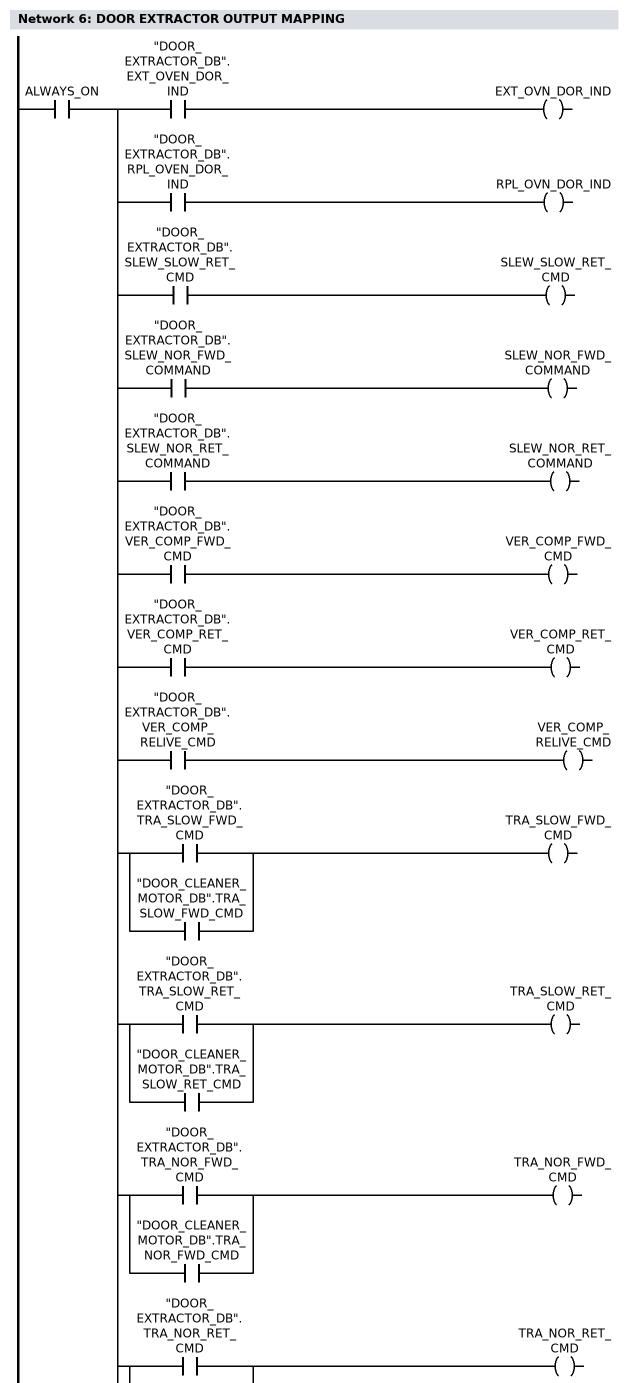
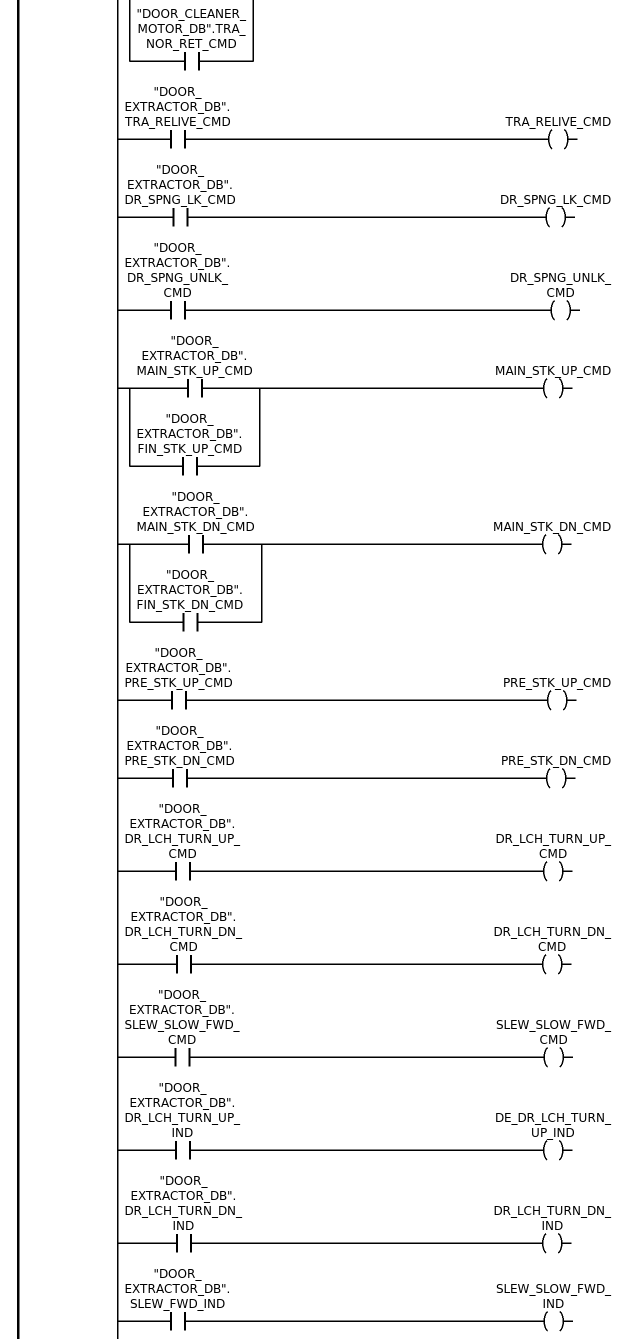
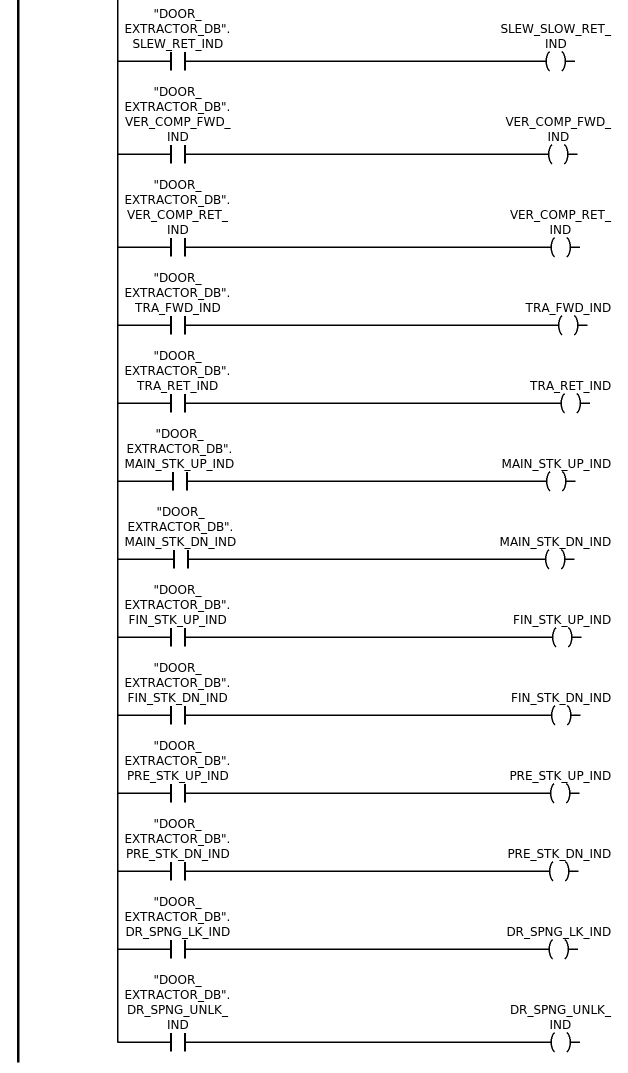
NETWORK
TITLE = DOOR EXTRACTOR OUTPUT MAPPING
//DOOR EXTRACTION
//
      A     "ALWAYS_ON";
      =     L 0.0;
      A     L 0.0;
      A     "DOOR_EXTRACTOR_DB".EXT_OVEN_DOR_IND;
      =     "EXT_OVN_DOR_IND";
      A     L 0.0;
      A     "DOOR_EXTRACTOR_DB".RPL_OVEN_DOR_IND;
      =     "RPL_OVN_DOR_IND";
      A     L 0.0;
      A     "DOOR_EXTRACTOR_DB".SLEW_SLOW_RET_CMD;
      =     "SLEW_SLOW_RET_CMD";
      A     L 0.0;
      A     "DOOR_EXTRACTOR_DB".SLEW_NOR_FWD_COMMAND;
      =     "SLEW_NOR_FWD_COMMAND";
      A     L 0.0;
      A     "DOOR_EXTRACTOR_DB".SLEW_NOR_RET_COMMAND;
      =     "SLEW_NOR_RET_COMMAND";
      A     L 0.0;
      A     "DOOR_EXTRACTOR_DB".VER_COMP_FWD_CMD;
      =     "VER_COMP_FWD_CMD";
      A     L 0.0;
      A     "DOOR_EXTRACTOR_DB".VER_COMP_RET_CMD;
      =     "VER_COMP_RET_CMD";
      A     L 0.0;
      A     "DOOR_EXTRACTOR_DB".VER_COMP_RELIVE_CMD;
      =     "VER_COMP_RELIVE_CMD";
      A     L 0.0;
      A(;
      O     "DOOR_EXTRACTOR_DB".TRA_SLOW_FWD_CMD;
      O     "DOOR_CLEANER_MOTOR_DB".TRA_SLOW_FWD_CMD;
      );
      =     "TRA_SLOW_FWD_CMD";
      A     L 0.0;
      A(;
      O     "DOOR_EXTRACTOR_DB".TRA_SLOW_RET_CMD;
      O     "DOOR_CLEANER_MOTOR_DB".TRA_SLOW_RET_CMD;
      );
      =     "TRA_SLOW_RET_CMD";
      A     L 0.0;
      A(;
      O     "DOOR_EXTRACTOR_DB".TRA_NOR_FWD_CMD;
      O     "DOOR_CLEANER_MOTOR_DB".TRA_NOR_FWD_CMD;
      );
      =     "TRA_NOR_FWD_CMD";
      A     L 0.0;
      A(;
      O     "DOOR_EXTRACTOR_DB".TRA_NOR_RET_CMD;
      O     "DOOR_CLEANER_MOTOR_DB".TRA_NOR_RET_CMD;
      );
      =     "TRA_NOR_RET_CMD";
      A     L 0.0;
      A     "DOOR_EXTRACTOR_DB".TRA_RELIVE_CMD;
      =     "TRA_RELIVE_CMD";
      A     L 0.0;
      A     "DOOR_EXTRACTOR_DB".DR_SPNG_LK_CMD;
      =     "DR_SPNG_LK_CMD";
      A     L 0.0;
      A     "DOOR_EXTRACTOR_DB".DR_SPNG_UNLK_CMD;
      =     "DR_SPNG_UNLK_CMD";
      A     L 0.0;
      A(;
      O     "DOOR_EXTRACTOR_DB".MAIN_STK_UP_CMD;
      O     "DOOR_EXTRACTOR_DB".FIN_STK_UP_CMD;
      );
      =     "MAIN_STK_UP_CMD";
      A     L 0.0;
      A(;
      O     "DOOR_EXTRACTOR_DB".MAIN_STK_DN_CMD;
      O     "DOOR_EXTRACTOR_DB".FIN_STK_DN_CMD;
      );
      =     "MAIN_STK_DN_CMD";
      A     L 0.0;
      A     "DOOR_EXTRACTOR_DB".PRE_STK_UP_CMD;
      =     "PRE_STK_UP_CMD";
      A     L 0.0;
      A     "DOOR_EXTRACTOR_DB".PRE_STK_DN_CMD;
      =     "PRE_STK_DN_CMD";
      A     L 0.0;
      A     "DOOR_EXTRACTOR_DB".DR_LCH_TURN_UP_CMD;
      =     "DR_LCH_TURN_UP_CMD";
      A     L 0.0;
      A     "DOOR_EXTRACTOR_DB".DR_LCH_TURN_DN_CMD;
      =     "DR_LCH_TURN_DN_CMD";
      A     L 0.0;
      A     "DOOR_EXTRACTOR_DB".SLEW_SLOW_FWD_CMD;
      =     "SLEW_SLOW_FWD_CMD";
      A     L 0.0;
      A     "DOOR_EXTRACTOR_DB".DR_LCH_TURN_UP_IND;
      =     "DE_DR_LCH_TURN_UP_IND";
      A     L 0.0;
      A     "DOOR_EXTRACTOR_DB".DR_LCH_TURN_DN_IND;
      =     "DR_LCH_TURN_DN_IND";
      A     L 0.0;
      A     "DOOR_EXTRACTOR_DB".SLEW_FWD_IND;
      =     "SLEW_SLOW_FWD_IND";
      A     L 0.0;
      A     "DOOR_EXTRACTOR_DB".SLEW_RET_IND;
      =     "SLEW_SLOW_RET_IND";
      A     L 0.0;
      A     "DOOR_EXTRACTOR_DB".VER_COMP_FWD_IND;
      =     "VER_COMP_FWD_IND";
      A     L 0.0;
      A     "DOOR_EXTRACTOR_DB".VER_COMP_RET_IND;
      =     "VER_COMP_RET_IND";
      A     L 0.0;
      A     "DOOR_EXTRACTOR_DB".TRA_FWD_IND;
      =     "TRA_FWD_IND";
      A     L 0.0;
      A     "DOOR_EXTRACTOR_DB".TRA_RET_IND;
      =     "TRA_RET_IND";
      A     L 0.0;
      A     "DOOR_EXTRACTOR_DB".MAIN_STK_UP_IND;
      =     "MAIN_STK_UP_IND";
      A     L 0.0;
      A     "DOOR_EXTRACTOR_DB".MAIN_STK_DN_IND;
      =     "MAIN_STK_DN_IND";
      A     L 0.0;
      A     "DOOR_EXTRACTOR_DB".FIN_STK_UP_IND;
      =     "FIN_STK_UP_IND";
      A     L 0.0;
      A     "DOOR_EXTRACTOR_DB".FIN_STK_DN_IND;
      =     "FIN_STK_DN_IND";
      A     L 0.0;
      A     "DOOR_EXTRACTOR_DB".PRE_STK_UP_IND;
      =     "PRE_STK_UP_IND";
      A     L 0.0;
      A     "DOOR_EXTRACTOR_DB".PRE_STK_DN_IND;
      =     "PRE_STK_DN_IND";
      A     L 0.0;
      A     "DOOR_EXTRACTOR_DB".DR_SPNG_LK_IND;
      =     "DR_SPNG_LK_IND";
      A     L 0.0;
      A     "DOOR_EXTRACTOR_DB".DR_SPNG_UNLK_IND;
      =     "DR_SPNG_UNLK_IND";
